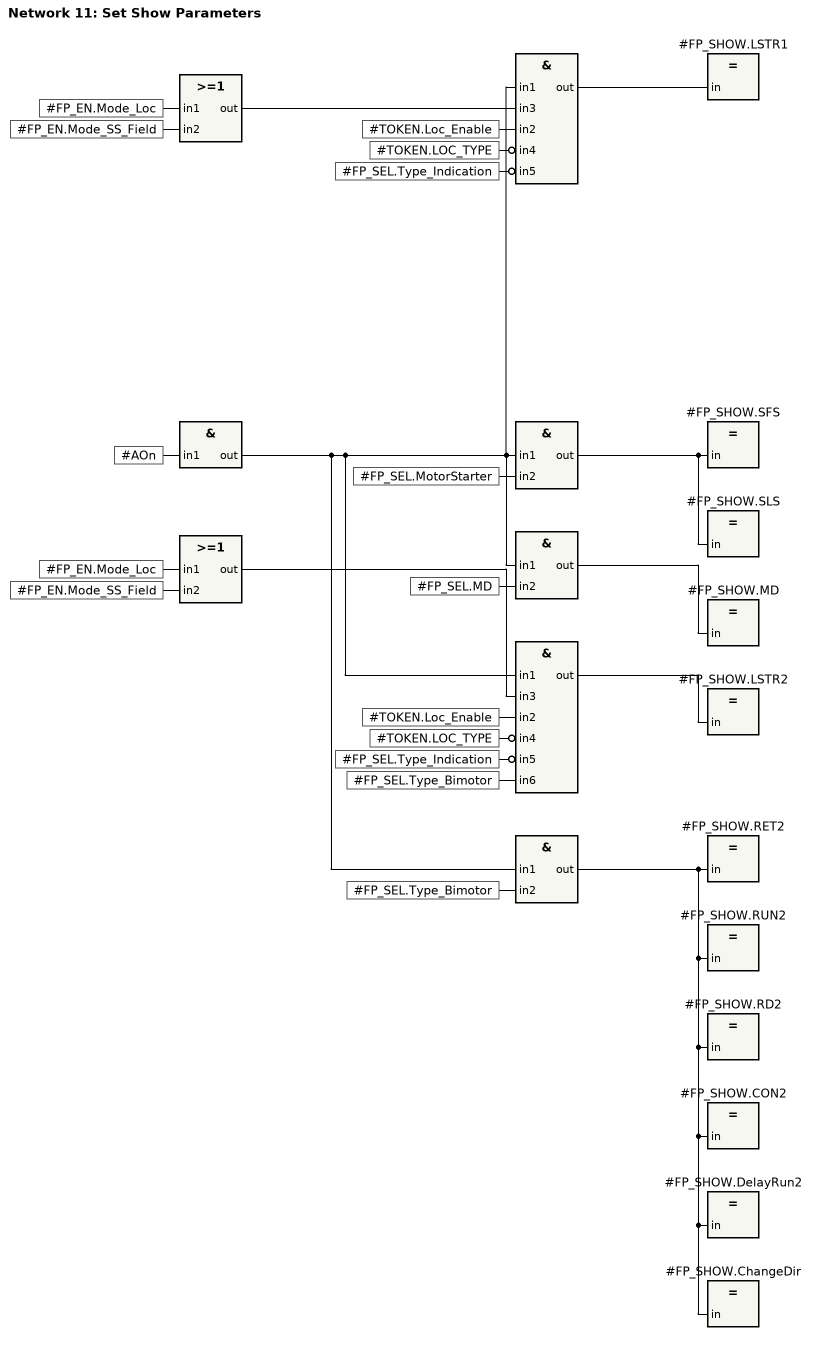
   #FP_SHOW.SFS := #AOn AND #FP_SEL.MotorStarter;
   #FP_SHOW.SLS := #FP_SHOW.SFS;
   #FP_SHOW.MD := #AOn AND #FP_SEL.MD;
   #FP_SHOW.LSTR1 := #AOn AND (#FP_EN.Mode_Loc OR #FP_EN.Mode_SS_Field) AND #TOKEN.Loc_Enable AND NOT #TOKEN.LOC_TYPE AND NOT #FP_SEL.Type_Indication;
   #FP_SHOW.LSTR2 := #AOn AND (#FP_EN.Mode_Loc OR #FP_EN.Mode_SS_Field) AND #TOKEN.Loc_Enable AND NOT #TOKEN.LOC_TYPE AND NOT #FP_SEL.Type_Indication AND #FP_SEL.Type_Bimotor;
   #FP_SHOW.RET2 := #AOn AND #FP_SEL.Type_Bimotor;
   #FP_SHOW.RUN2 := #FP_SHOW.RET2;
   #FP_SHOW.RD2 := #FP_SHOW.RET2;
   #FP_SHOW.CON2 := #FP_SHOW.RET2;
   #FP_SHOW.DelayRun2 := #FP_SHOW.RET2;
   #FP_SHOW.ChangeDir := #FP_SHOW.RET2;
END_REGION

REGION Network 12: SELECT
   // Build 003 - 1.July.2019 (EXTBOB): Added logic to prevent group selection interference when motor is running in "electrical" local mode or mode is controlled from the field.
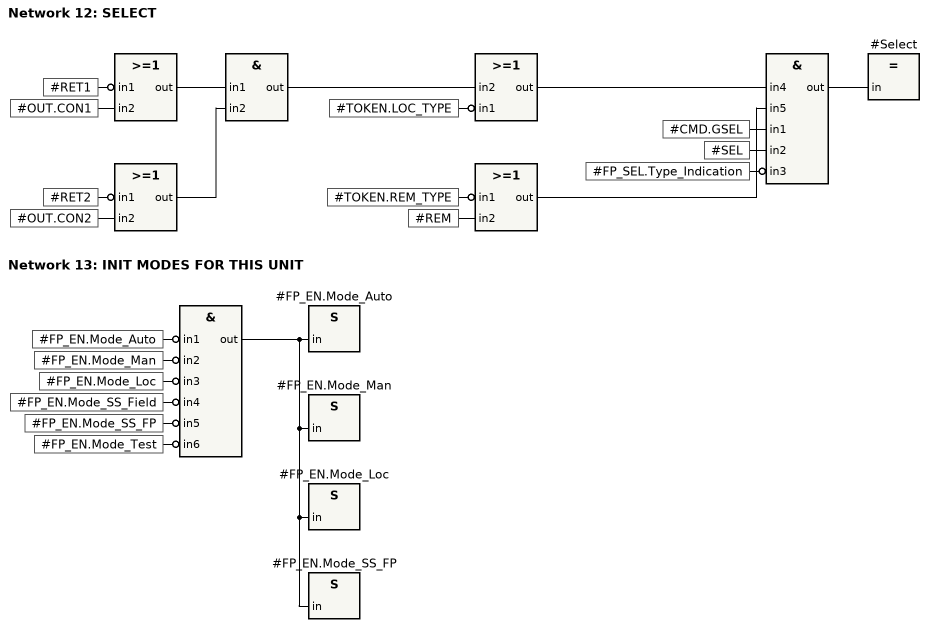
   #Select := (((NOT #RET1 OR #OUT.CON1) AND (NOT #RET2 OR #OUT.CON2)) OR NOT #TOKEN.LOC_TYPE) AND (NOT #TOKEN.REM_TYPE OR #REM) AND #CMD.GSEL AND #SEL AND NOT #FP_SEL.Type_Indication;
END_REGION

REGION Network 13: INIT MODES FOR THIS UNIT
   #_w1 := NOT #FP_EN.Mode_Auto AND NOT #FP_EN.Mode_Man AND NOT #FP_EN.Mode_Loc AND NOT #FP_EN.Mode_SS_Field AND NOT #FP_EN.Mode_SS_FP AND NOT #FP_EN.Mode_Test;
   IF #_w1 THEN
       #FP_EN.Mode_Auto := TRUE;
       #FP_EN.Mode_Man := TRUE;
       #FP_EN.Mode_Loc := TRUE;
       #FP_EN.Mode_SS_FP := TRUE;
   END_IF;
END_REGION

REGION Network 14: SHOW PUSH BUTTONS ON FACEPLATE
   // Build 002 - 25 March 2019 : Loc_type flag removed from Show_Local flag
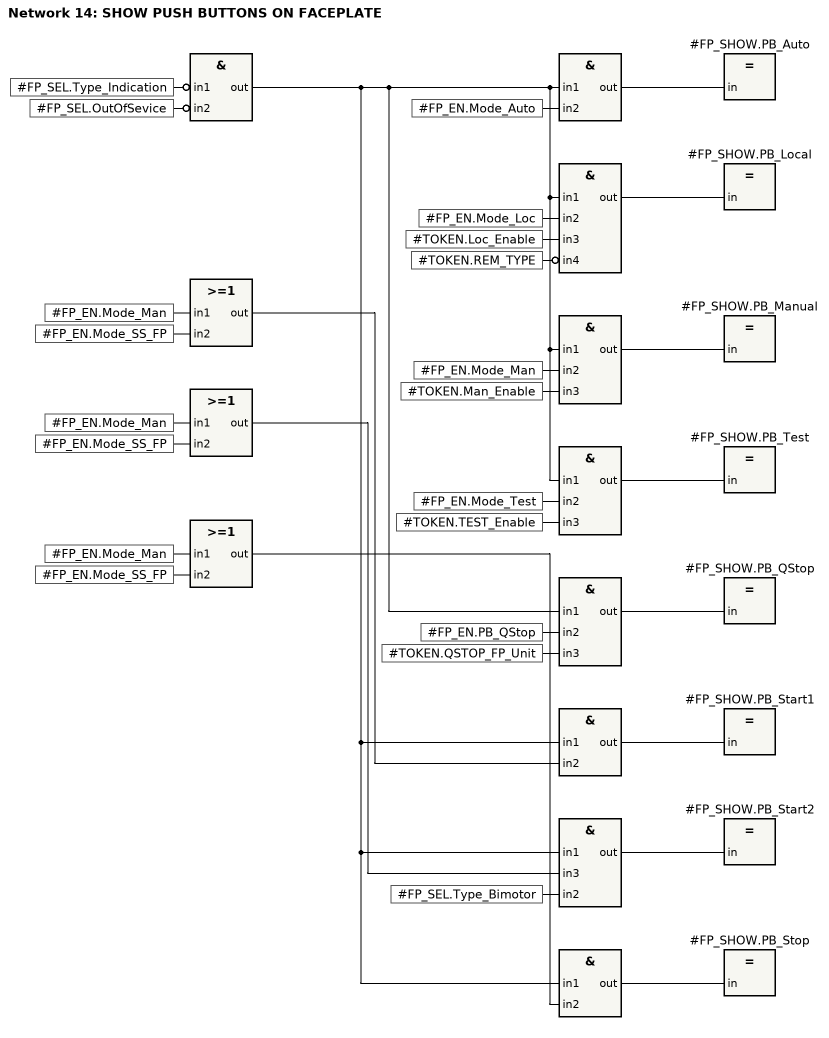
   #_w1 := NOT #FP_SEL.Type_Indication AND NOT #FP_SEL.OutOfSevice;
   #FP_SHOW.PB_Auto := #_w1 AND #FP_EN.Mode_Auto;
   #FP_SHOW.PB_Local := #_w1 AND #FP_EN.Mode_Loc AND #TOKEN.Loc_Enable AND NOT #TOKEN.REM_TYPE;
   #FP_SHOW.PB_Manual := #_w1 AND #FP_EN.Mode_Man AND #TOKEN.Man_Enable;
   #FP_SHOW.PB_Test := #_w1 AND #FP_EN.Mode_Test AND #TOKEN.TEST_Enable;
   #FP_SHOW.PB_QStop := #_w1 AND #FP_EN.PB_QStop AND #TOKEN.QSTOP_FP_Unit;
   #FP_SHOW.PB_Start1 := #_w1 AND (#FP_EN.Mode_Man OR #FP_EN.Mode_SS_FP);
   #FP_SHOW.PB_Start2 := #_w1 AND (#FP_EN.Mode_Man OR #FP_EN.Mode_SS_FP) AND #FP_SEL.Type_Bimotor;
   #FP_SHOW.PB_Stop := #_w1 AND (#FP_EN.Mode_Man OR #FP_EN.Mode_SS_FP);
END_REGION

REGION Network 15: DIMOUT AUTO BUTTON ON FACEPLATE
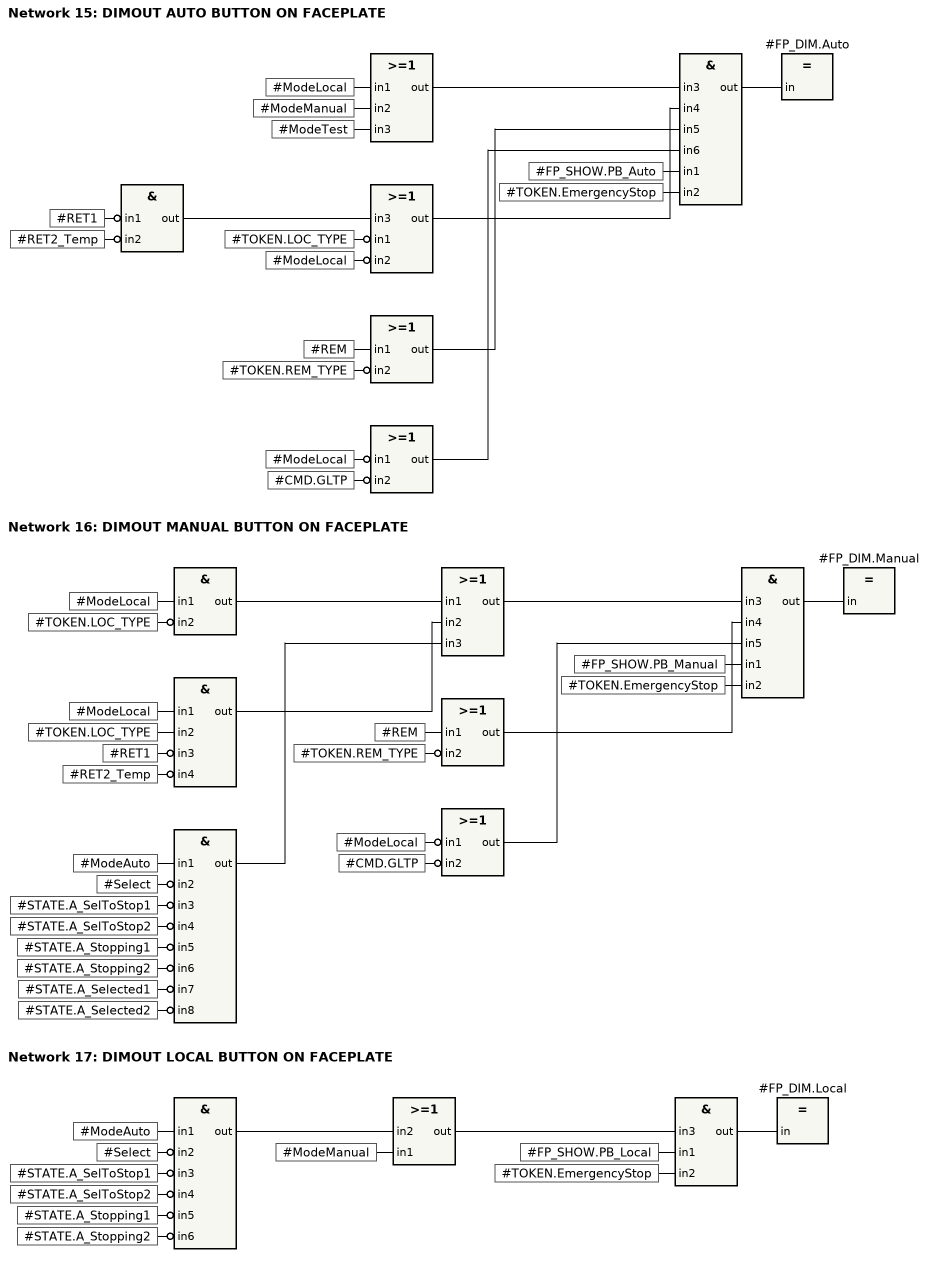
   #FP_DIM.Auto := (#ModeLocal OR #ModeManual OR #ModeTest) AND ((NOT #RET1 AND NOT #RET2_Temp) OR NOT #TOKEN.LOC_TYPE OR NOT #ModeLocal) AND (#REM OR NOT #TOKEN.REM_TYPE) AND (NOT #ModeLocal OR NOT #CMD.GLTP) AND #FP_SHOW.PB_Auto AND #TOKEN.EmergencyStop;
END_REGION

REGION Network 16: DIMOUT MANUAL BUTTON ON FACEPLATE
   #FP_DIM.Manual := ((#ModeLocal AND NOT #TOKEN.LOC_TYPE) OR (#ModeLocal AND #TOKEN.LOC_TYPE AND NOT #RET1 AND NOT #RET2_Temp) OR (#ModeAuto AND NOT #Select AND NOT #STATE.A_SelToStop1 AND NOT #STATE.A_SelToStop2 AND NOT #STATE.A_Stopping1 AND NOT #STATE.A_Stopping2 AND NOT #STATE.A_Selected1 AND NOT #STATE.A_Selected2)) AND (#REM OR NOT #TOKEN.REM_TYPE) AND (NOT #ModeLocal OR NOT #CMD.GLTP) AND #FP_SHOW.PB_Manual AND #TOKEN.EmergencyStop;
END_REGION

REGION Network 17: DIMOUT LOCAL BUTTON ON FACEPLATE
   #FP_DIM.Local := ((#ModeAuto AND NOT #Select AND NOT #STATE.A_SelToStop1 AND NOT #STATE.A_SelToStop2 AND NOT #STATE.A_Stopping1 AND NOT #STATE.A_Stopping2) OR #ModeManual) AND #FP_SHOW.PB_Local AND #TOKEN.EmergencyStop;
END_REGION

REGION Network 18: DIMOUT TEST BUTTON ON FACEPLATE
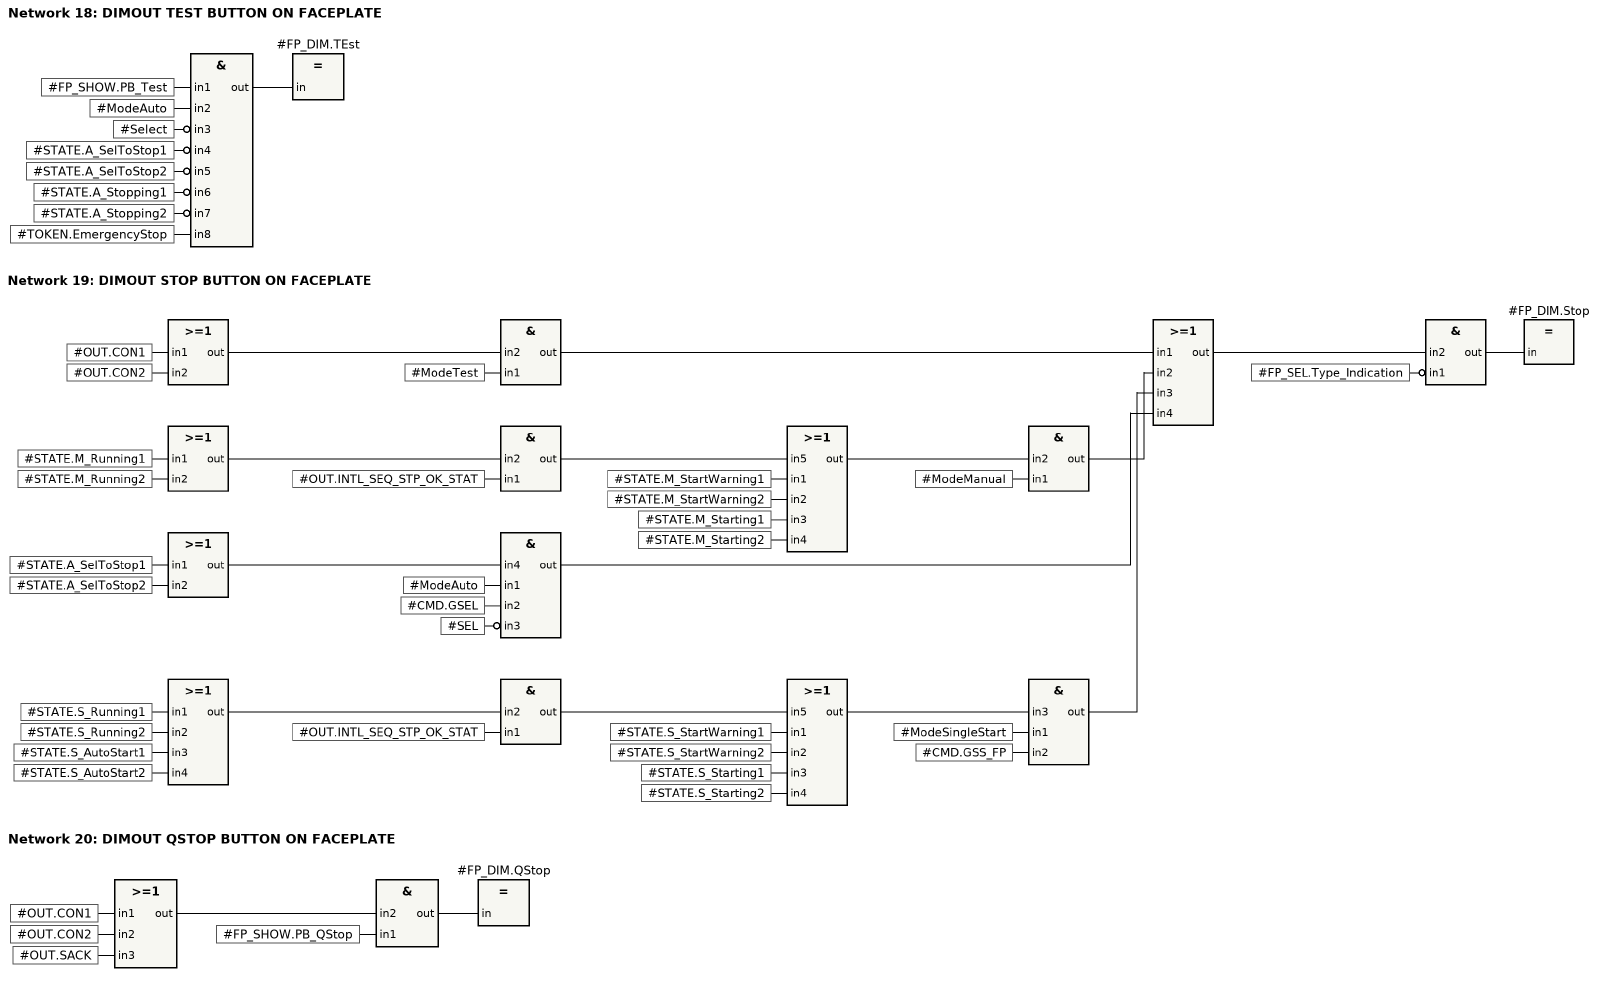
   #FP_DIM.TEst := #FP_SHOW.PB_Test AND #ModeAuto AND NOT #Select AND NOT #STATE.A_SelToStop1 AND NOT #STATE.A_SelToStop2 AND NOT #STATE.A_Stopping1 AND NOT #STATE.A_Stopping2 AND #TOKEN.EmergencyStop;
END_REGION

REGION Network 19: DIMOUT STOP BUTTON ON FACEPLATE
   #FP_DIM.Stop := (((#OUT.CON1 OR #OUT.CON2) AND #ModeTest) OR ((((#STATE.M_Running1 OR #STATE.M_Running2) AND #OUT.INTL_SEQ_STP_OK_STAT) OR #STATE.M_StartWarning1 OR #STATE.M_StartWarning2 OR #STATE.M_Starting1 OR #STATE.M_Starting2) AND #ModeManual) OR ((((#STATE.S_Running1 OR #STATE.S_Running2 OR #STATE.S_AutoStart1 OR #STATE.S_AutoStart2) AND #OUT.INTL_SEQ_STP_OK_STAT) OR #STATE.S_StartWarning1 OR #STATE.S_StartWarning2 OR #STATE.S_Starting1 OR #STATE.S_Starting2) AND #ModeSingleStart AND #CMD.GSS_FP) OR ((#STATE.A_SelToStop1 OR #STATE.A_SelToStop2) AND #ModeAuto AND #CMD.GSEL AND NOT #SEL)) AND NOT #FP_SEL.Type_Indication;
END_REGION

REGION Network 20: DIMOUT QSTOP BUTTON ON FACEPLATE
   #FP_DIM.QStop := (#OUT.CON1 OR #OUT.CON2 OR #OUT.SACK) AND #FP_SHOW.PB_QStop;
END_REGION

REGION Network 21: DIMOUT START1 BUTTON ON FACEPLATE
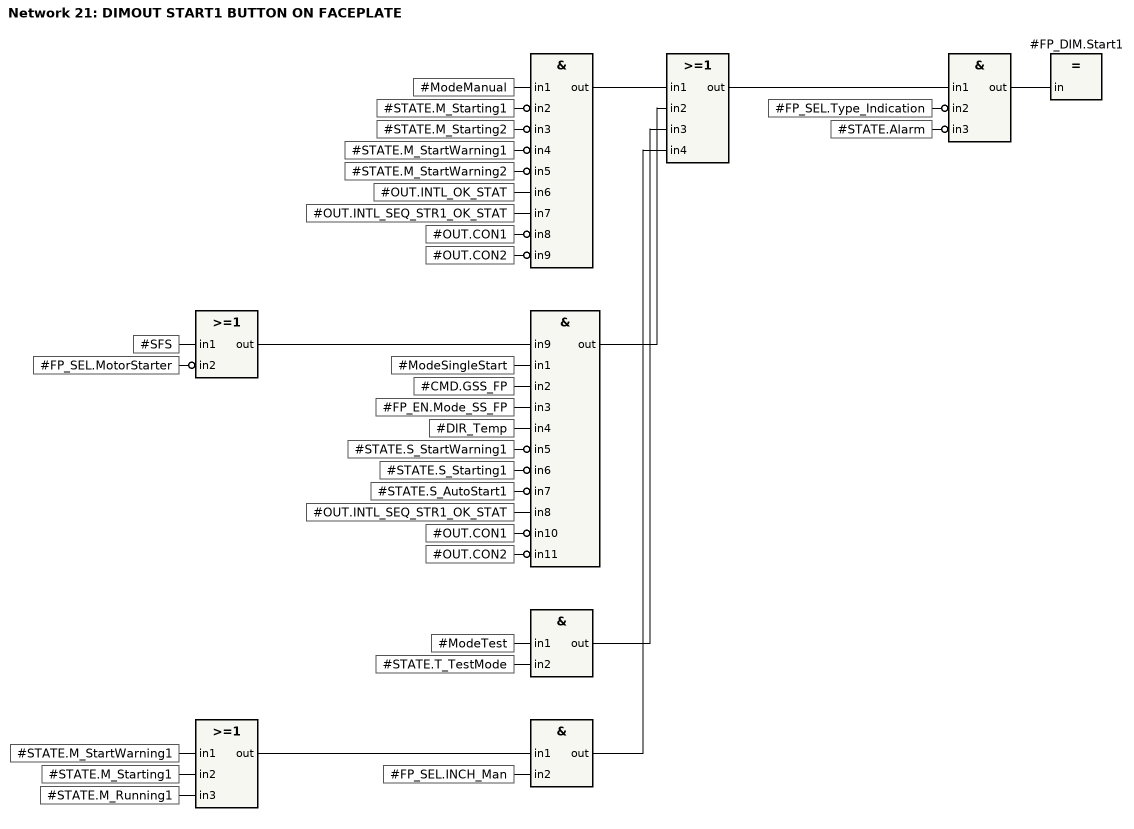
   #FP_DIM.Start1 := ((#ModeManual AND NOT #STATE.M_Starting1 AND NOT #STATE.M_Starting2 AND NOT #STATE.M_StartWarning1 AND NOT #STATE.M_StartWarning2 AND #OUT.INTL_OK_STAT AND #OUT.INTL_SEQ_STR1_OK_STAT AND NOT #OUT.CON1 AND NOT #OUT.CON2) OR ((#SFS OR NOT #FP_SEL.MotorStarter) AND #ModeSingleStart AND #CMD.GSS_FP AND #FP_EN.Mode_SS_FP AND #DIR_Temp AND NOT #STATE.S_StartWarning1 AND NOT #STATE.S_Starting1 AND NOT #STATE.S_AutoStart1 AND #OUT.INTL_SEQ_STR1_OK_STAT AND NOT #OUT.CON1 AND NOT #OUT.CON2) OR (#ModeTest AND #STATE.T_TestMode) OR ((#STATE.M_StartWarning1 OR #STATE.M_Starting1 OR #STATE.M_Running1) AND #FP_SEL.INCH_Man)) AND NOT #FP_SEL.Type_Indication AND NOT #STATE.Alarm;
END_REGION

REGION Network 22: DIMOUT START2 BUTTON ON FACEPLATE
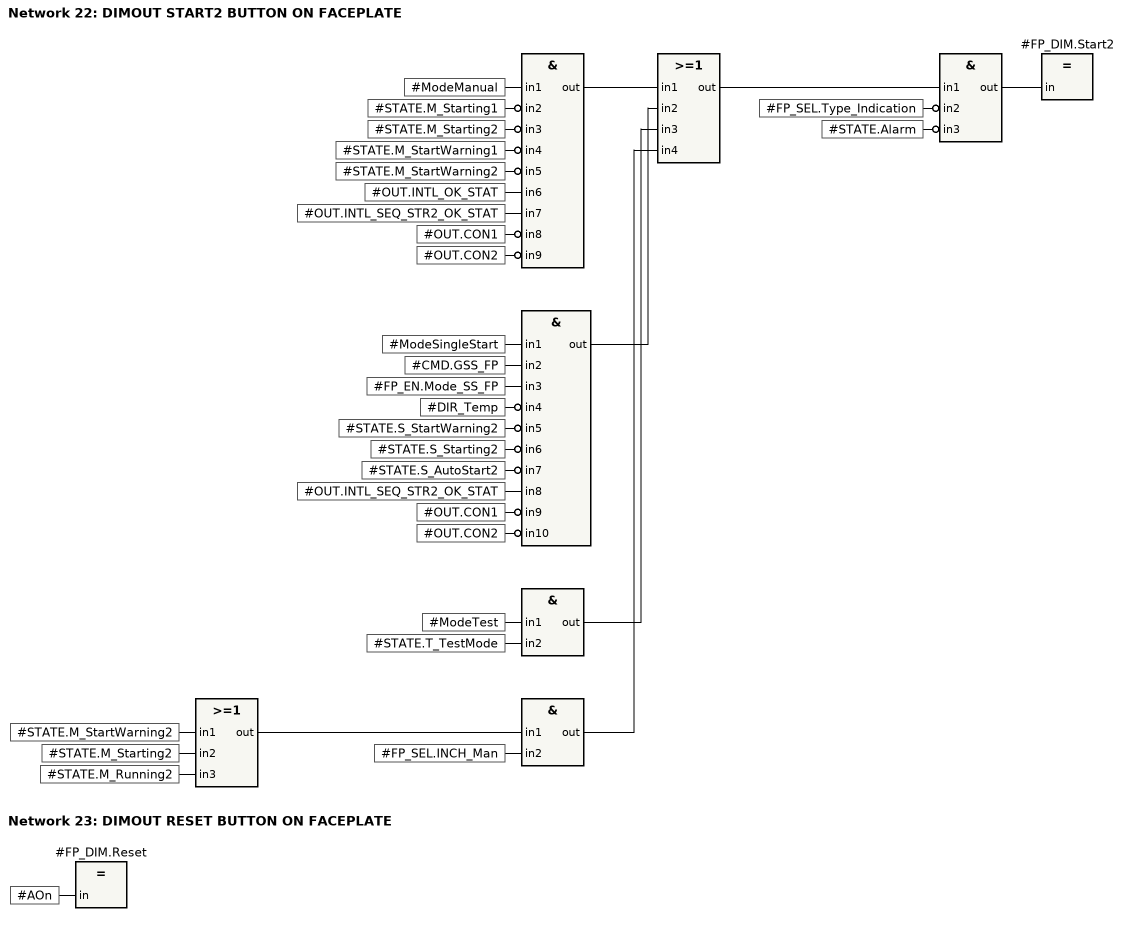
   #FP_DIM.Start2 := ((#ModeManual AND NOT #STATE.M_Starting1 AND NOT #STATE.M_Starting2 AND NOT #STATE.M_StartWarning1 AND NOT #STATE.M_StartWarning2 AND #OUT.INTL_OK_STAT AND #OUT.INTL_SEQ_STR2_OK_STAT AND NOT #OUT.CON1 AND NOT #OUT.CON2) OR (#ModeSingleStart AND #CMD.GSS_FP AND #FP_EN.Mode_SS_FP AND NOT #DIR_Temp AND NOT #STATE.S_StartWarning2 AND NOT #STATE.S_Starting2 AND NOT #STATE.S_AutoStart2 AND #OUT.INTL_SEQ_STR2_OK_STAT AND NOT #OUT.CON1 AND NOT #OUT.CON2) OR (#ModeTest AND #STATE.T_TestMode) OR ((#STATE.M_StartWarning2 OR #STATE.M_Starting2 OR #STATE.M_Running2) AND #FP_SEL.INCH_Man)) AND NOT #FP_SEL.Type_Indication AND NOT #STATE.Alarm;
END_REGION

REGION Network 23: DIMOUT RESET BUTTON ON FACEPLATE
   #FP_DIM.Reset := #AOn;
END_REGION

REGION Network 24: Auto Mode
   // Build 002 - 25 March 2019 : REM flag removed from Modelocal FP_CMD_Auto command
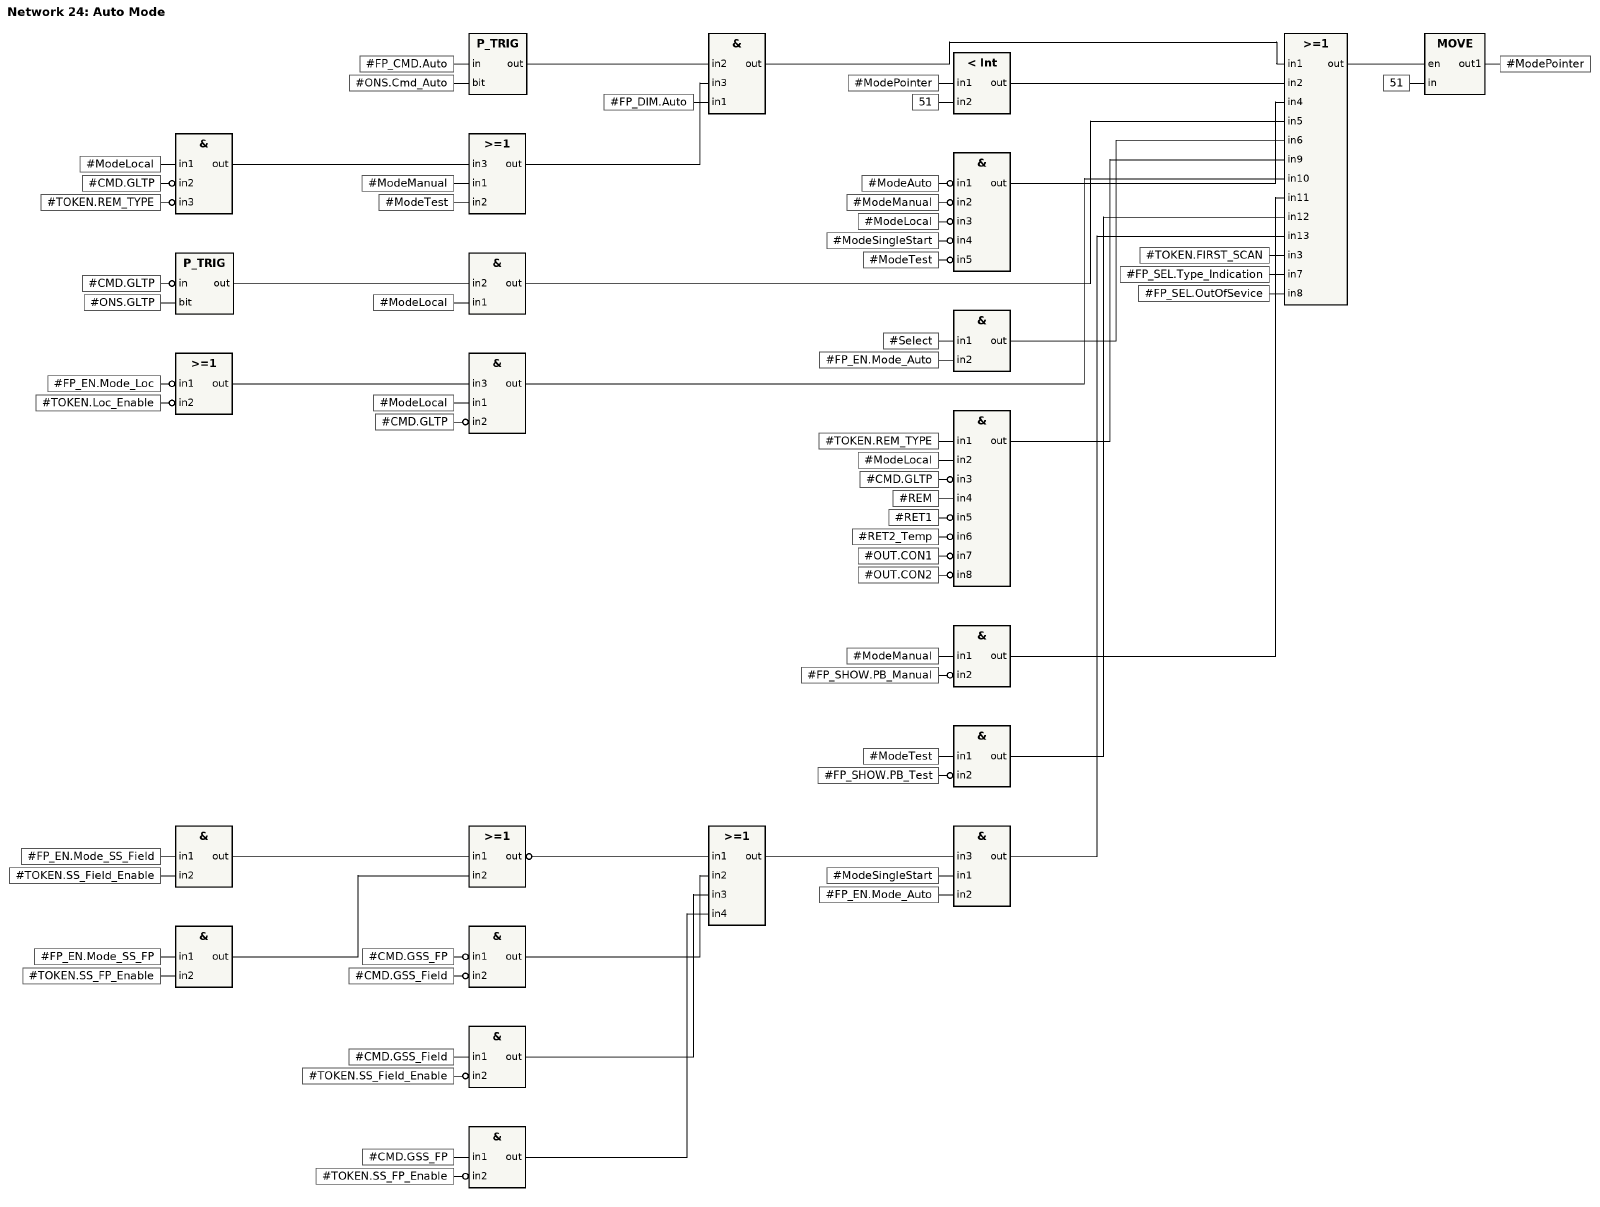
   #_w1 := #FP_CMD.Auto AND NOT #ONS.Cmd_Auto;   // rising edge
   #ONS.Cmd_Auto := #FP_CMD.Auto;
   #_w2 := NOT #CMD.GLTP AND NOT #ONS.GLTP;   // rising edge
   #ONS.GLTP := NOT #CMD.GLTP;
   IF (#_w1 AND ((#ModeLocal AND NOT #CMD.GLTP AND NOT #TOKEN.REM_TYPE) OR #ModeManual OR #ModeTest) AND #FP_DIM.Auto) OR (#ModePointer < 51) OR (NOT #ModeAuto AND NOT #ModeManual AND NOT #ModeLocal AND NOT #ModeSingleStart AND NOT #ModeTest) OR (#_w2 AND #ModeLocal) OR (#Select AND #FP_EN.Mode_Auto) OR (#TOKEN.REM_TYPE AND #ModeLocal AND NOT #CMD.GLTP AND #REM AND NOT #RET1 AND NOT #RET2_Temp AND NOT #OUT.CON1 AND NOT #OUT.CON2) OR ((NOT #FP_EN.Mode_Loc OR NOT #TOKEN.Loc_Enable) AND #ModeLocal AND NOT #CMD.GLTP) OR (#ModeManual AND NOT #FP_SHOW.PB_Manual) OR (#ModeTest AND NOT #FP_SHOW.PB_Test) OR ((NOT ((#FP_EN.Mode_SS_Field AND #TOKEN.SS_Field_Enable) OR (#FP_EN.Mode_SS_FP AND #TOKEN.SS_FP_Enable)) OR (NOT #CMD.GSS_FP AND NOT #CMD.GSS_Field) OR (#CMD.GSS_Field AND NOT #TOKEN.SS_Field_Enable) OR (#CMD.GSS_FP AND NOT #TOKEN.SS_FP_Enable)) AND #ModeSingleStart AND #FP_EN.Mode_Auto) OR #TOKEN.FIRST_SCAN OR #FP_SEL.Type_Indication OR #FP_SEL.OutOfSevice THEN
       #ModePointer := 51;
   END_IF;
END_REGION

REGION Network 25: Mode Manual
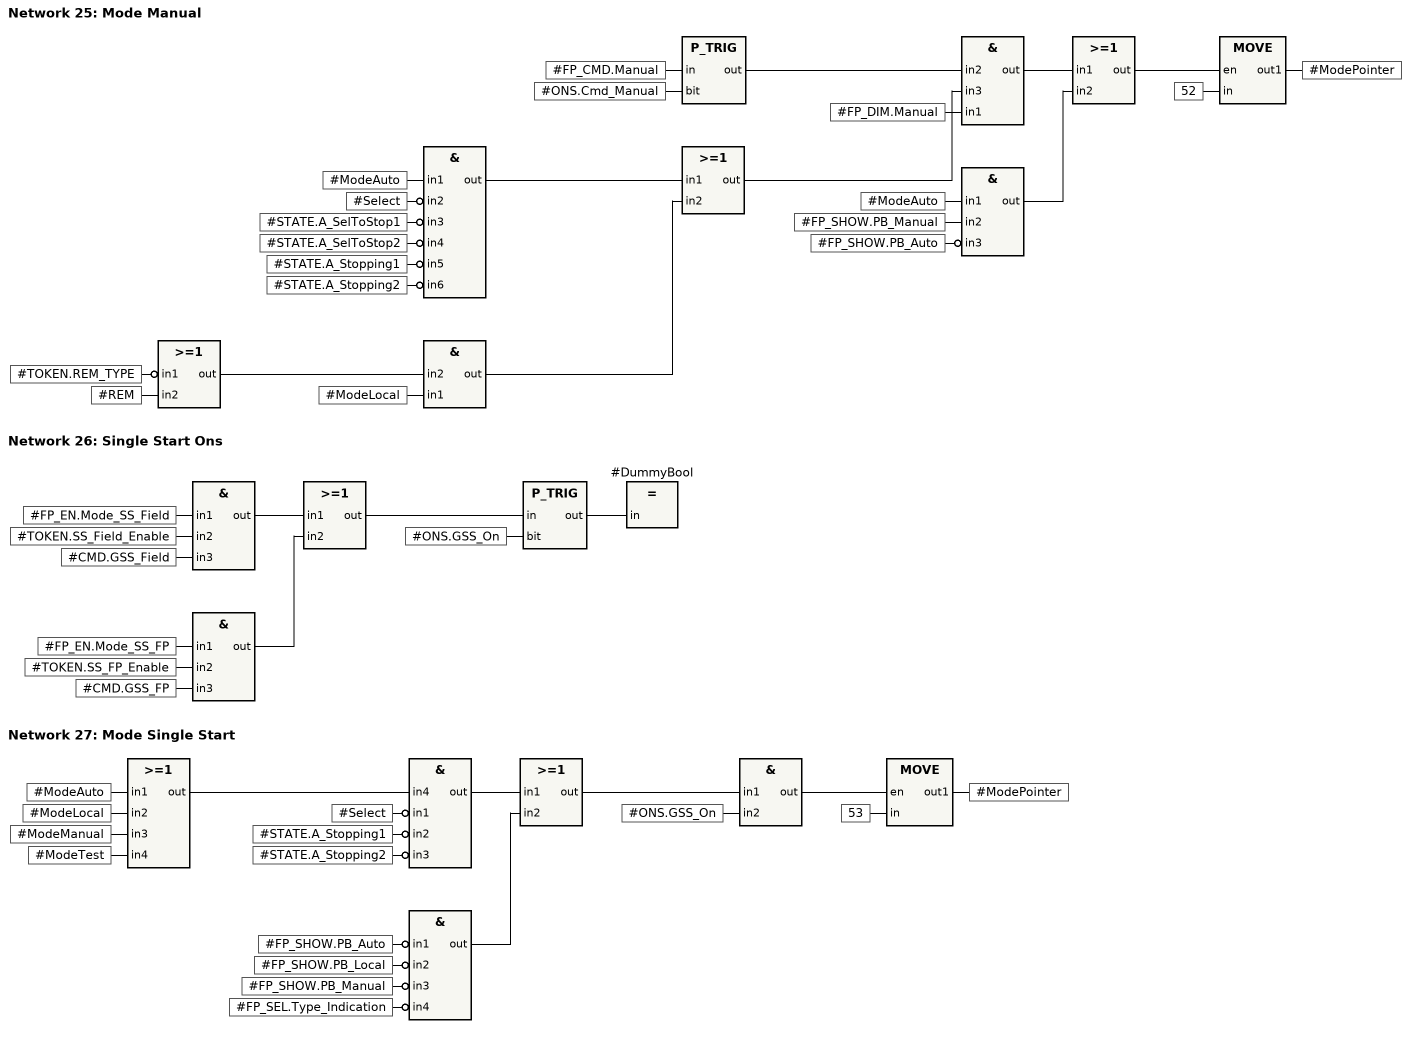
   #_w1 := #FP_CMD.Manual AND NOT #ONS.Cmd_Manual;   // rising edge
   #ONS.Cmd_Manual := #FP_CMD.Manual;
   IF (#_w1 AND ((#ModeAuto AND NOT #Select AND NOT #STATE.A_SelToStop1 AND NOT #STATE.A_SelToStop2 AND NOT #STATE.A_Stopping1 AND NOT #STATE.A_Stopping2) OR ((NOT #TOKEN.REM_TYPE OR #REM) AND #ModeLocal)) AND #FP_DIM.Manual) OR (#ModeAuto AND #FP_SHOW.PB_Manual AND NOT #FP_SHOW.PB_Auto) THEN
       #ModePointer := 52;
   END_IF;
END_REGION

REGION Network 26: Single Start Ons
   // Build 003 - 1.July.2019 (EXTBOB): Added ONS and Created New Network to separate trigger from pre-conditions
   #_w1 := (#FP_EN.Mode_SS_Field AND #TOKEN.SS_Field_Enable AND #CMD.GSS_Field) OR (#FP_EN.Mode_SS_FP AND #TOKEN.SS_FP_Enable AND #CMD.GSS_FP);
   #_w2 := #_w1 AND NOT #ONS.GSS_On;   // rising edge
   #ONS.GSS_On := #_w1;
   #DummyBool := #_w2;
END_REGION

REGION Network 27: Mode Single Start
   // Build 003 - 1.July.2019 (EXTBOB): Added Single Start ONS and Removed the Single start trigger condition & made as seperate Network above
   IF (((#ModeAuto OR #ModeLocal OR #ModeManual OR #ModeTest) AND NOT #Select AND NOT #STATE.A_Stopping1 AND NOT #STATE.A_Stopping2) OR (NOT #FP_SHOW.PB_Auto AND NOT #FP_SHOW.PB_Local AND NOT #FP_SHOW.PB_Manual AND NOT #FP_SEL.Type_Indication)) AND #ONS.GSS_On THEN
       #ModePointer := 53;
   END_IF;
END_REGION

REGION Network 28: Mode Local
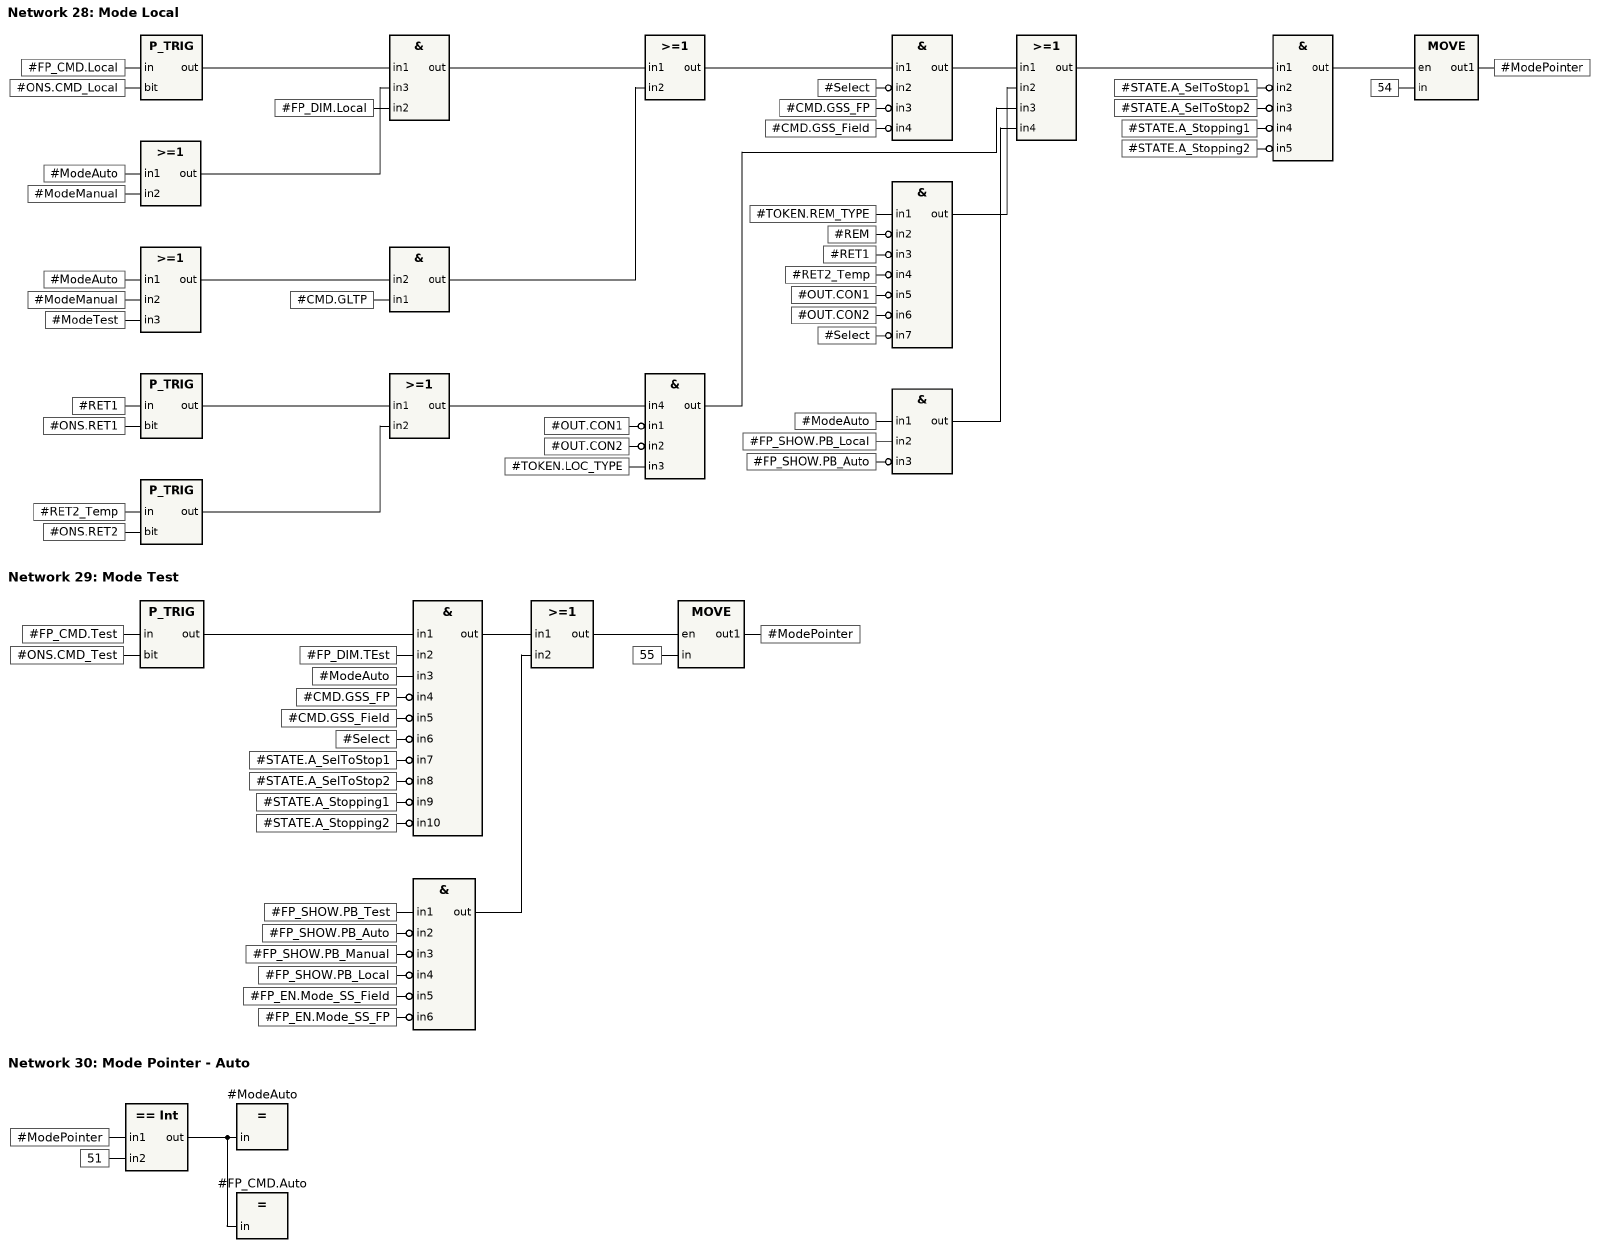
   #_w1 := #FP_CMD.Local AND NOT #ONS.CMD_Local;   // rising edge
   #ONS.CMD_Local := #FP_CMD.Local;
   #_w2 := #RET1 AND NOT #ONS.RET1;   // rising edge
   #ONS.RET1 := #RET1;
   #_w3 := #RET2_Temp AND NOT #ONS.RET2;   // rising edge
   #ONS.RET2 := #RET2_Temp;
   IF ((((#_w1 AND (#ModeAuto OR #ModeManual) AND #FP_DIM.Local) OR ((#ModeAuto OR #ModeManual OR #ModeTest) AND #CMD.GLTP)) AND NOT #Select AND NOT #CMD.GSS_FP AND NOT #CMD.GSS_Field) OR (#TOKEN.REM_TYPE AND NOT #REM AND NOT #RET1 AND NOT #RET2_Temp AND NOT #OUT.CON1 AND NOT #OUT.CON2 AND NOT #Select) OR ((#_w2 OR #_w3) AND NOT #OUT.CON1 AND NOT #OUT.CON2 AND #TOKEN.LOC_TYPE) OR (#ModeAuto AND #FP_SHOW.PB_Local AND NOT #FP_SHOW.PB_Auto)) AND NOT #STATE.A_SelToStop1 AND NOT #STATE.A_SelToStop2 AND NOT #STATE.A_Stopping1 AND NOT #STATE.A_Stopping2 THEN
       #ModePointer := 54;
   END_IF;
END_REGION

REGION Network 29: Mode Test
   #_w1 := #FP_CMD.Test AND NOT #ONS.CMD_Test;   // rising edge
   #ONS.CMD_Test := #FP_CMD.Test;
   IF (#_w1 AND #FP_DIM.TEst AND #ModeAuto AND NOT #CMD.GSS_FP AND NOT #CMD.GSS_Field AND NOT #Select AND NOT #STATE.A_SelToStop1 AND NOT #STATE.A_SelToStop2 AND NOT #STATE.A_Stopping1 AND NOT #STATE.A_Stopping2) OR (#FP_SHOW.PB_Test AND NOT #FP_SHOW.PB_Auto AND NOT #FP_SHOW.PB_Manual AND NOT #FP_SHOW.PB_Local AND NOT #FP_EN.Mode_SS_Field AND NOT #FP_EN.Mode_SS_FP) THEN
       #ModePointer := 55;
   END_IF;
END_REGION

REGION Network 30: Mode Pointer - Auto
   #ModeAuto := #ModePointer = 51;
   #FP_CMD.Auto := #ModeAuto;
END_REGION

REGION Network 31: Mode Pointer - Manual
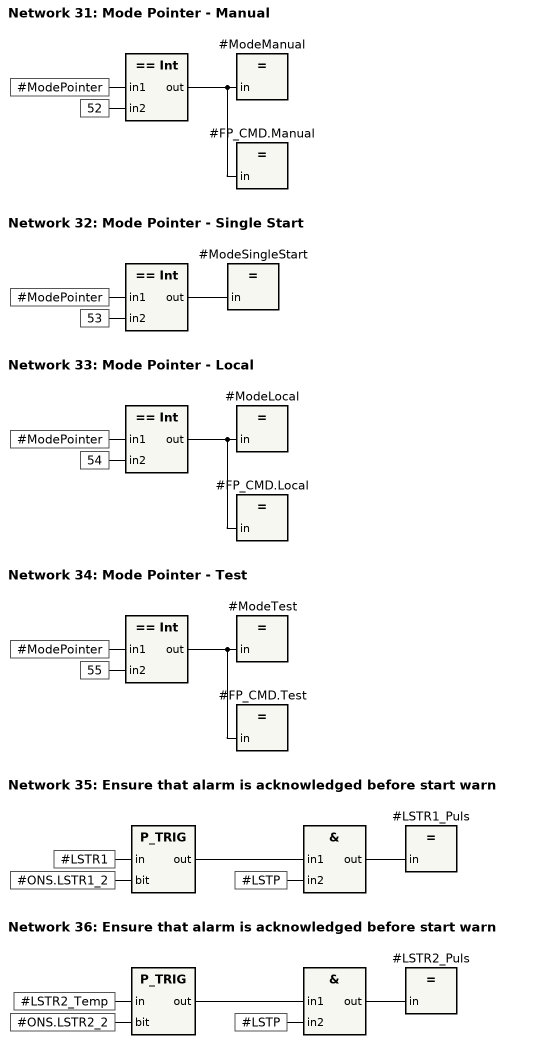
   #ModeManual := #ModePointer = 52;
   #FP_CMD.Manual := #ModeManual;
END_REGION

REGION Network 32: Mode Pointer - Single Start
   #ModeSingleStart := #ModePointer = 53;
END_REGION

REGION Network 33: Mode Pointer - Local
   #ModeLocal := #ModePointer = 54;
   #FP_CMD.Local := #ModeLocal;
END_REGION

REGION Network 34: Mode Pointer - Test
   #ModeTest := #ModePointer = 55;
   #FP_CMD.Test := #ModeTest;
END_REGION

REGION Network 35: Ensure that alarm is acknowledged before start warn
   // Build 003 - 30 Jun 2019 (EXTBOB): Added LSTP to prevent pulse output
   #_w1 := #LSTR1 AND NOT #ONS.LSTR1_2;   // rising edge
   #ONS.LSTR1_2 := #LSTR1;
   #LSTR1_Puls := #_w1 AND #LSTP;
END_REGION

REGION Network 36: Ensure that alarm is acknowledged before start warn
   // Build 003 - 30 Jun 2019 (EXTBOB): Added LSTP to prevent pulse output
   #_w1 := #LSTR2_Temp AND NOT #ONS.LSTR2_2;   // rising edge
   #ONS.LSTR2_2 := #LSTR2_Temp;
   #LSTR2_Puls := #_w1 AND #LSTP;
END_REGION

REGION Network 37: FACEPLATE COMMANDS (Pulse Type)
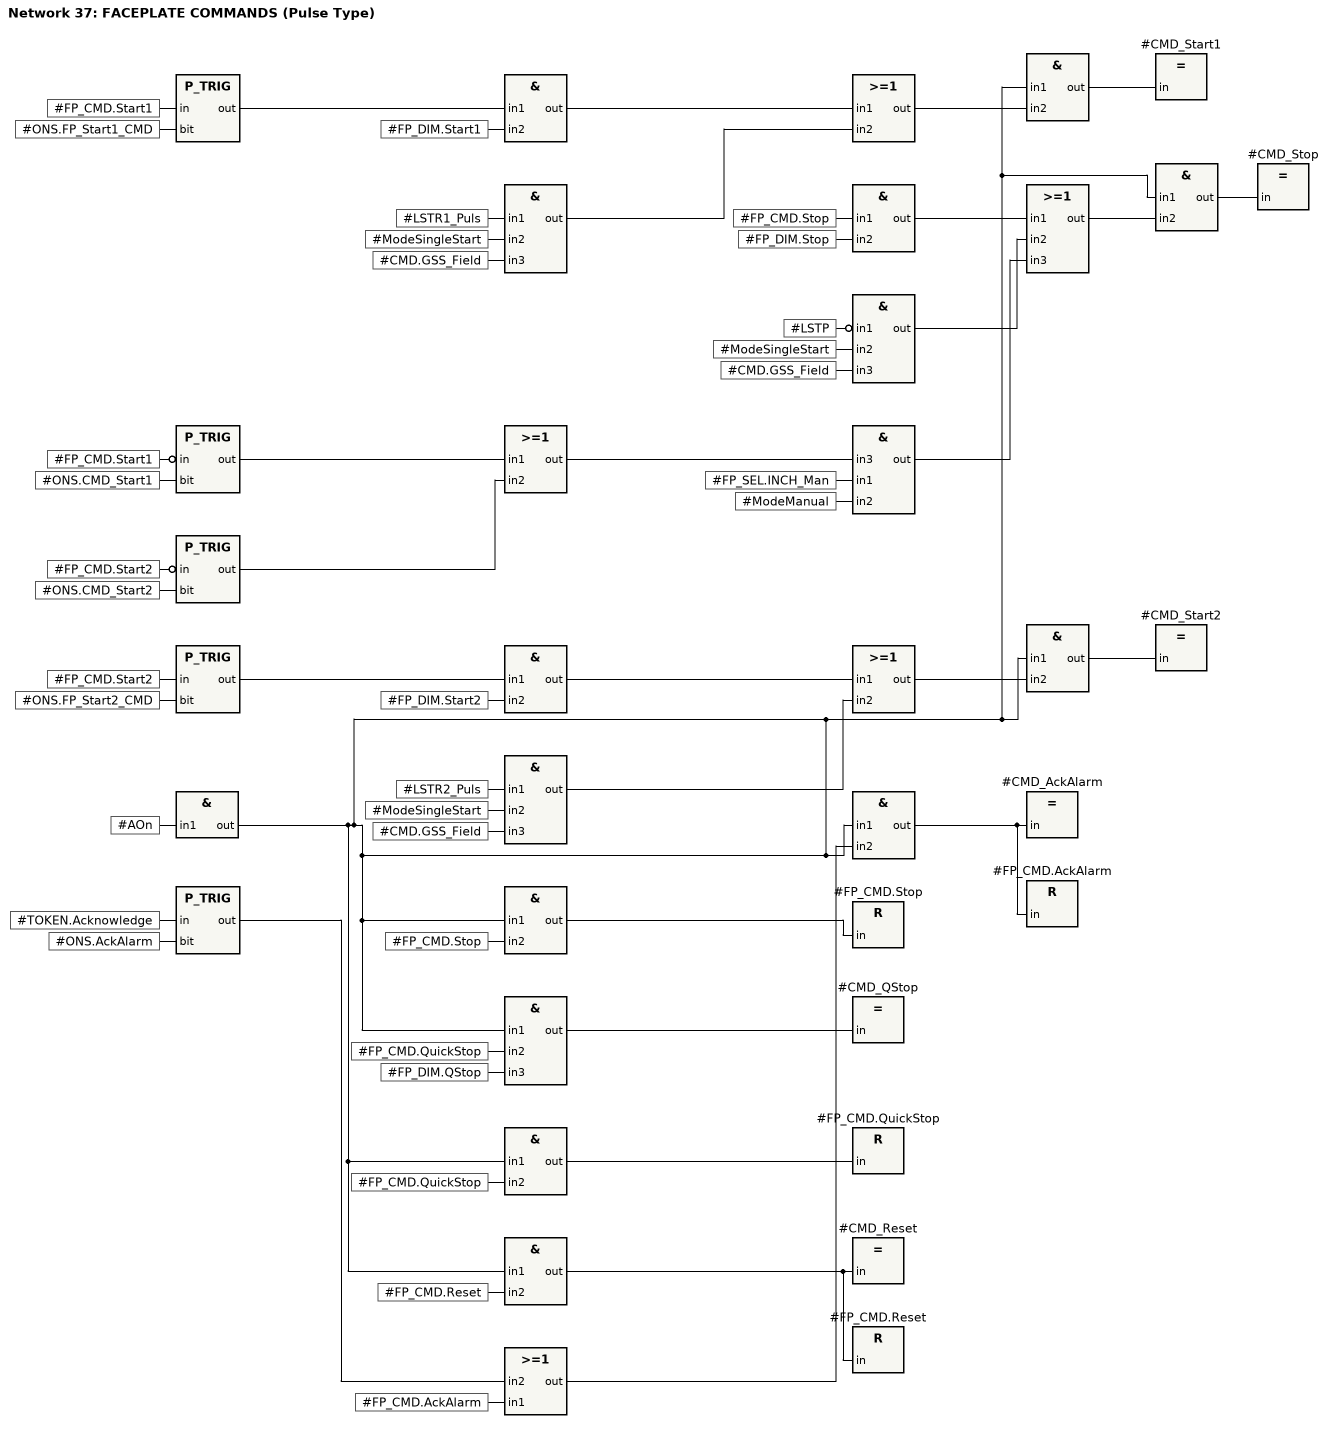
   #_w1 := #FP_CMD.Start1 AND NOT #ONS.FP_Start1_CMD;   // rising edge
   #ONS.FP_Start1_CMD := #FP_CMD.Start1;
   #CMD_Start1 := #AOn AND ((#_w1 AND #FP_DIM.Start1) OR (#LSTR1_Puls AND #ModeSingleStart AND #CMD.GSS_Field));
   #_w2 := #FP_CMD.Start2 AND NOT #ONS.FP_Start2_CMD;   // rising edge
   #ONS.FP_Start2_CMD := #FP_CMD.Start2;
   #CMD_Start2 := #AOn AND ((#_w2 AND #FP_DIM.Start2) OR (#LSTR2_Puls AND #ModeSingleStart AND #CMD.GSS_Field));
   #_w3 := NOT #FP_CMD.Start1 AND NOT #ONS.CMD_Start1;   // rising edge
   #ONS.CMD_Start1 := NOT #FP_CMD.Start1;
   #_w4 := NOT #FP_CMD.Start2 AND NOT #ONS.CMD_Start2;   // rising edge
   #ONS.CMD_Start2 := NOT #FP_CMD.Start2;
   #CMD_Stop := #AOn AND ((#FP_CMD.Stop AND #FP_DIM.Stop) OR (NOT #LSTP AND #ModeSingleStart AND #CMD.GSS_Field) OR ((#_w3 OR #_w4) AND #FP_SEL.INCH_Man AND #ModeManual));
   IF #AOn AND #FP_CMD.Stop THEN #FP_CMD.Stop := FALSE; END_IF;
   #CMD_QStop := #AOn AND #FP_CMD.QuickStop AND #FP_DIM.QStop;
   IF #AOn AND #FP_CMD.QuickStop THEN #FP_CMD.QuickStop := FALSE; END_IF;
   #CMD_Reset := #AOn AND #FP_CMD.Reset;
   IF #CMD_Reset THEN #FP_CMD.Reset := FALSE; END_IF;
   #_w5 := #TOKEN.Acknowledge AND NOT #ONS.AckAlarm;   // rising edge
   #ONS.AckAlarm := #TOKEN.Acknowledge;
   #CMD_AckAlarm := #AOn AND (#_w5 OR #FP_CMD.AckAlarm);
   IF #CMD_AckAlarm THEN #FP_CMD.AckAlarm := FALSE; END_IF;
END_REGION

REGION Network 38: Command Reset
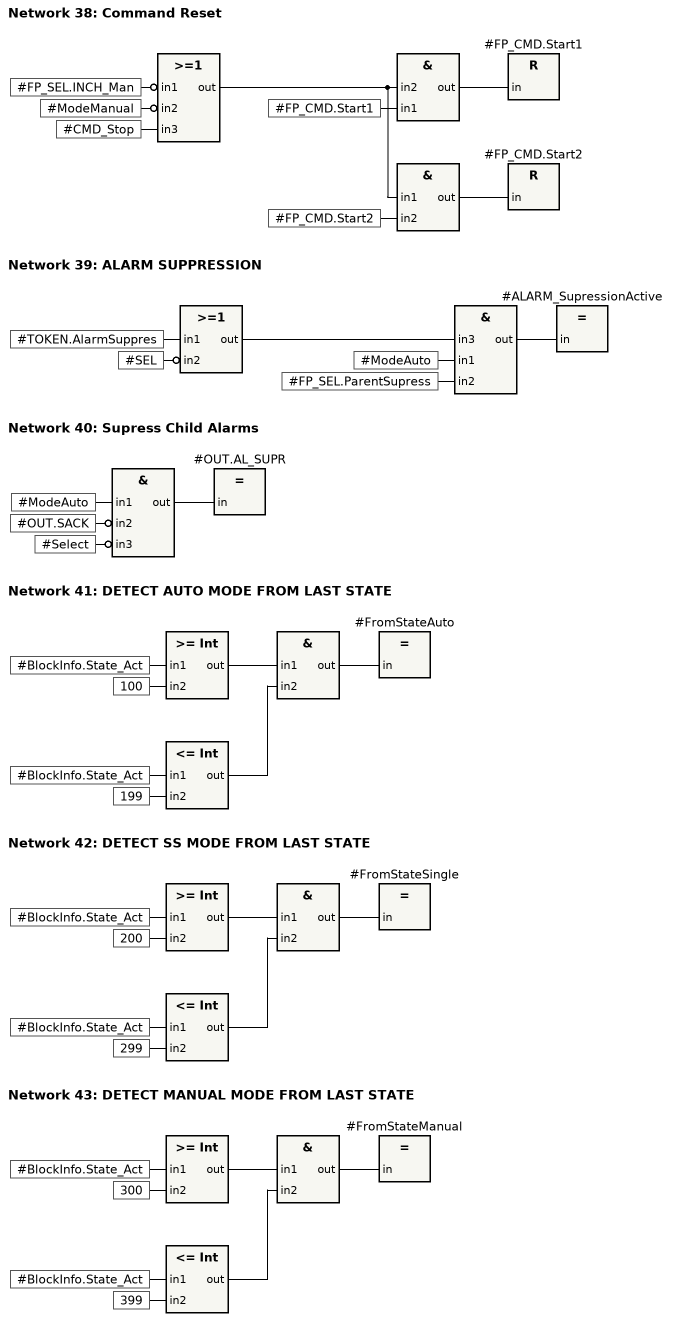
   #_w1 := NOT #FP_SEL.INCH_Man OR NOT #ModeManual OR #CMD_Stop;
   IF #_w1 AND #FP_CMD.Start1 THEN #FP_CMD.Start1 := FALSE; END_IF;
   IF #_w1 AND #FP_CMD.Start2 THEN #FP_CMD.Start2 := FALSE; END_IF;
END_REGION

REGION Network 39: ALARM SUPPRESSION
   #ALARM_SupressionActive := (#TOKEN.AlarmSuppres OR NOT #SEL) AND #ModeAuto AND #FP_SEL.ParentSupress;
END_REGION

REGION Network 40: Supress Child Alarms
   #OUT.AL_SUPR := #ModeAuto AND NOT #OUT.SACK AND NOT #Select;
END_REGION

REGION Network 41: DETECT AUTO MODE FROM LAST STATE
   #FromStateAuto := (#BlockInfo.State_Act >= 100) AND (#BlockInfo.State_Act <= 199);
END_REGION

REGION Network 42: DETECT SS MODE FROM LAST STATE
   #FromStateSingle := (#BlockInfo.State_Act >= 200) AND (#BlockInfo.State_Act <= 299);
END_REGION

REGION Network 43: DETECT MANUAL MODE FROM LAST STATE
   #FromStateManual := (#BlockInfo.State_Act >= 300) AND (#BlockInfo.State_Act <= 399);
END_REGION

REGION Network 44: DETECT LOCAL MODE FROM LAST STATE
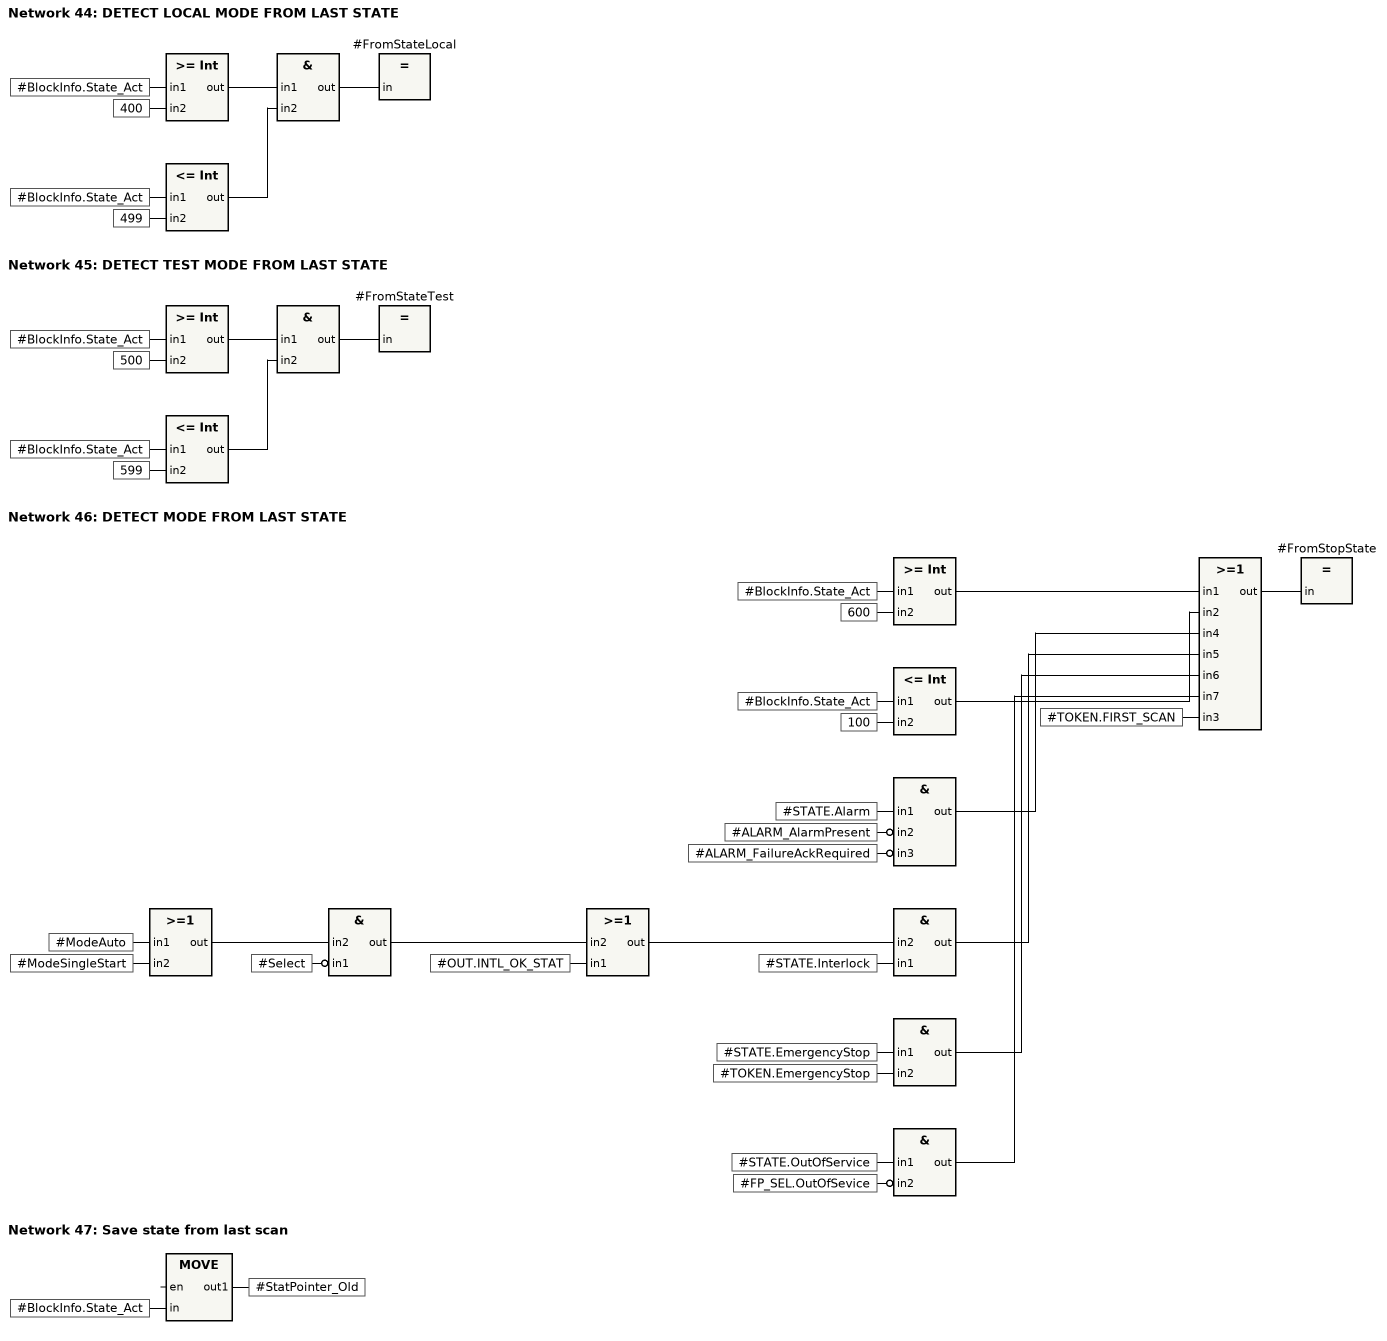
   #FromStateLocal := (#BlockInfo.State_Act >= 400) AND (#BlockInfo.State_Act <= 499);
END_REGION

REGION Network 45: DETECT TEST MODE FROM LAST STATE
   #FromStateTest := (#BlockInfo.State_Act >= 500) AND (#BlockInfo.State_Act <= 599);
END_REGION

REGION Network 46: DETECT MODE FROM LAST STATE
   #FromStopState := (#BlockInfo.State_Act >= 600) OR (#BlockInfo.State_Act <= 100) OR (#STATE.Alarm AND NOT #ALARM_AlarmPresent AND NOT #ALARM_FailureAckRequired) OR ((((#ModeAuto OR #ModeSingleStart) AND NOT #Select) OR #OUT.INTL_OK_STAT) AND #STATE.Interlock) OR (#STATE.EmergencyStop AND #TOKEN.EmergencyStop) OR (#STATE.OutOfService AND NOT #FP_SEL.OutOfSevice) OR #TOKEN.FIRST_SCAN;
END_REGION

REGION Network 47: Save state from last scan
   #StatPointer_Old := #BlockInfo.State_Act;
END_REGION

REGION Network 48
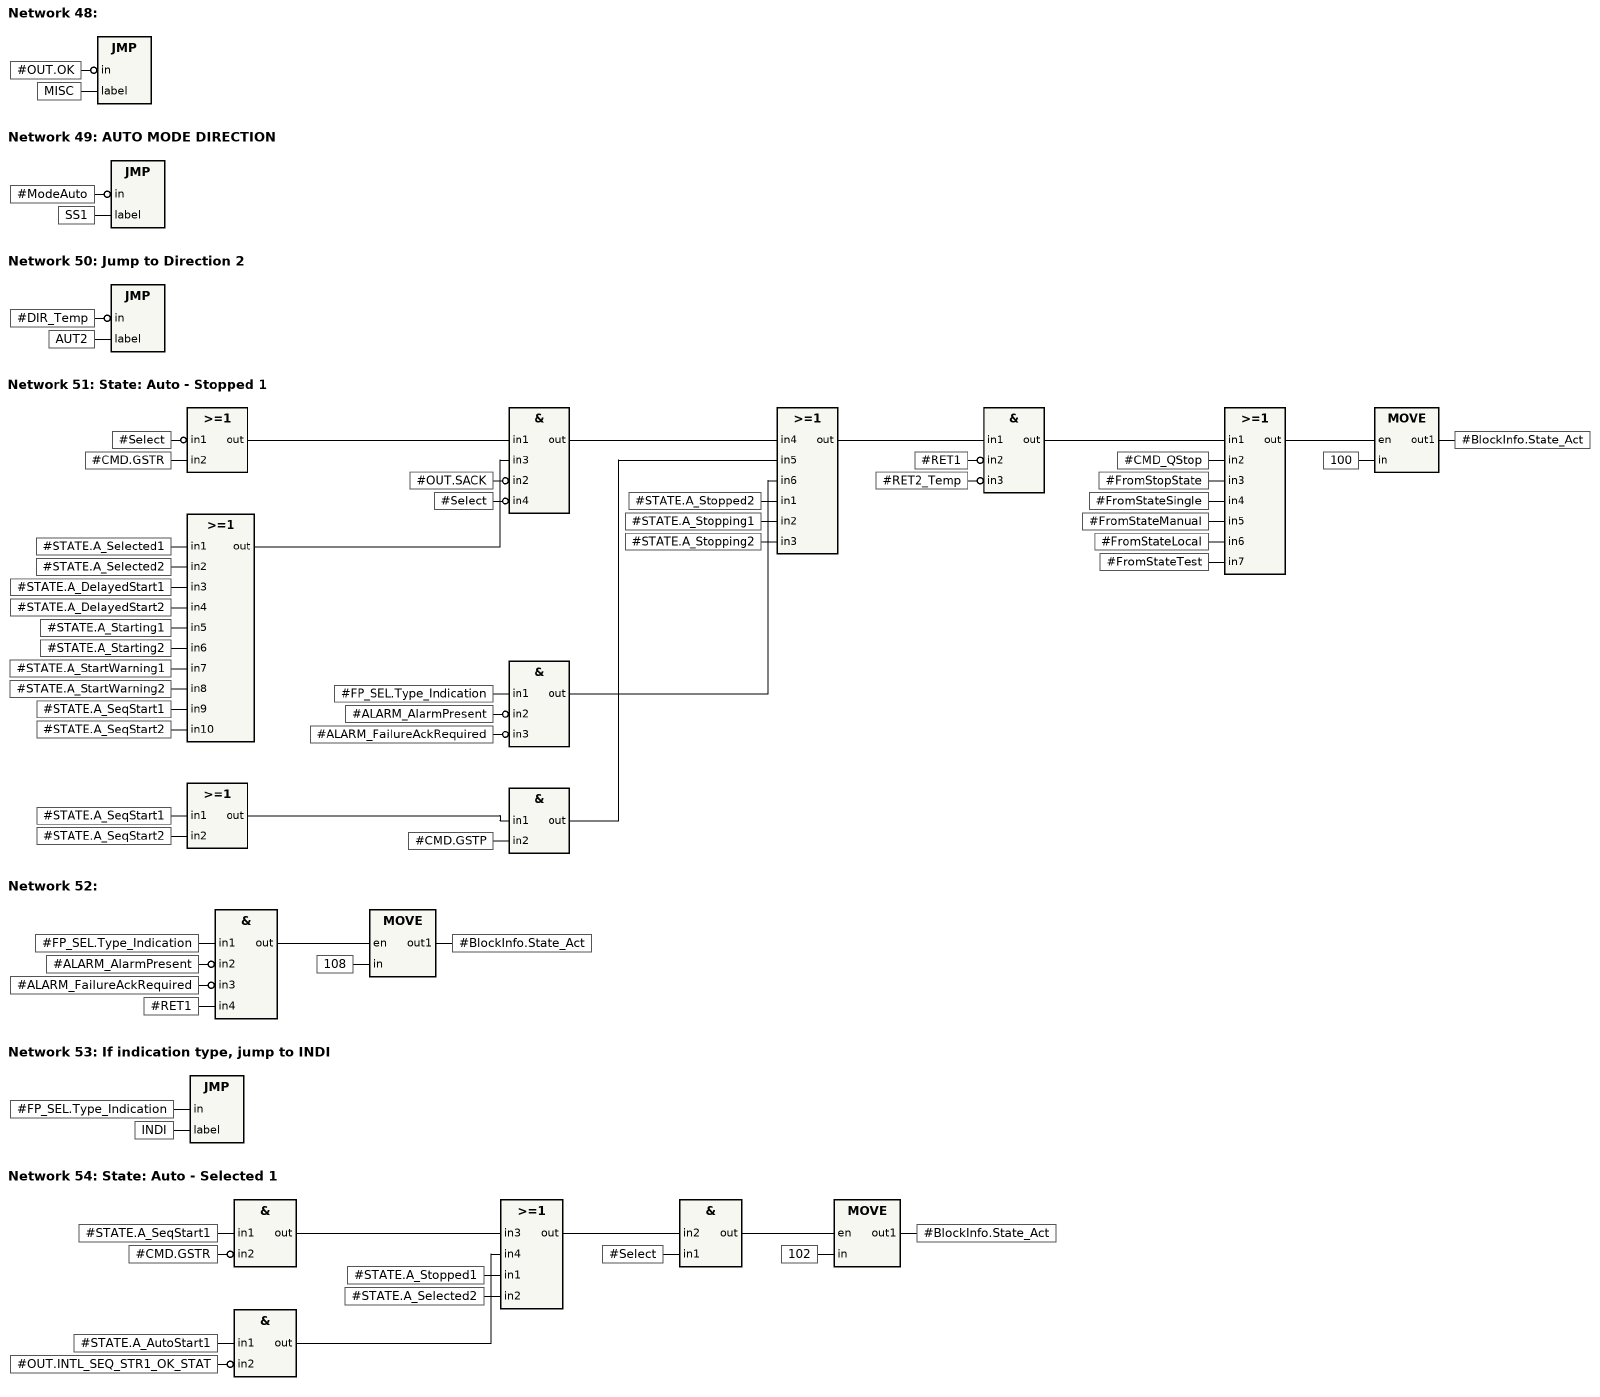
   IF NOT #OUT.OK THEN GOTO MISC; END_IF;
END_REGION

REGION Network 49: AUTO MODE DIRECTION
   IF NOT #ModeAuto THEN GOTO SS1; END_IF;
END_REGION

REGION Network 50: Jump to Direction 2
   IF NOT #DIR_Temp THEN GOTO AUT2; END_IF;
END_REGION

REGION Network 51: State: Auto - Stopped 1
   IF ((((NOT #Select OR #CMD.GSTR) AND (#STATE.A_Selected1 OR #STATE.A_Selected2 OR #STATE.A_DelayedStart1 OR #STATE.A_DelayedStart2 OR #STATE.A_Starting1 OR #STATE.A_Starting2 OR #STATE.A_StartWarning1 OR #STATE.A_StartWarning2 OR #STATE.A_SeqStart1 OR #STATE.A_SeqStart2) AND NOT #OUT.SACK AND NOT #Select) OR ((#STATE.A_SeqStart1 OR #STATE.A_SeqStart2) AND #CMD.GSTP) OR (#FP_SEL.Type_Indication AND NOT #ALARM_AlarmPresent AND NOT #ALARM_FailureAckRequired) OR #STATE.A_Stopped2 OR #STATE.A_Stopping1 OR #STATE.A_Stopping2) AND NOT #RET1 AND NOT #RET2_Temp) OR #CMD_QStop OR #FromStopState OR #FromStateSingle OR #FromStateManual OR #FromStateLocal OR #FromStateTest THEN
       #BlockInfo.State_Act := 100;
   END_IF;
END_REGION

REGION Network 52
   IF #FP_SEL.Type_Indication AND NOT #ALARM_AlarmPresent AND NOT #ALARM_FailureAckRequired AND #RET1 THEN
       #BlockInfo.State_Act := 108;
   END_IF;
END_REGION

REGION Network 53: If indication type, jump to INDI
   IF #FP_SEL.Type_Indication THEN GOTO INDI; END_IF;
END_REGION

REGION Network 54: State: Auto - Selected 1
   // Build 002 - 25 March 2019 : AutoStart1 with SeqStart Interlock condition added
   IF ((#STATE.A_SeqStart1 AND NOT #CMD.GSTR) OR (#STATE.A_AutoStart1 AND NOT #OUT.INTL_SEQ_STR1_OK_STAT) OR #STATE.A_Stopped1 OR #STATE.A_Selected2) AND #Select THEN
       #BlockInfo.State_Act := 102;
   END_IF;
END_REGION

REGION Network 55: State: Auto - Sequence Start 1
   // Build 006 - 29 Aug 2019 (EXTBOB) : AutoStart flag removed to have wait start state when astr = 0 during group start contion
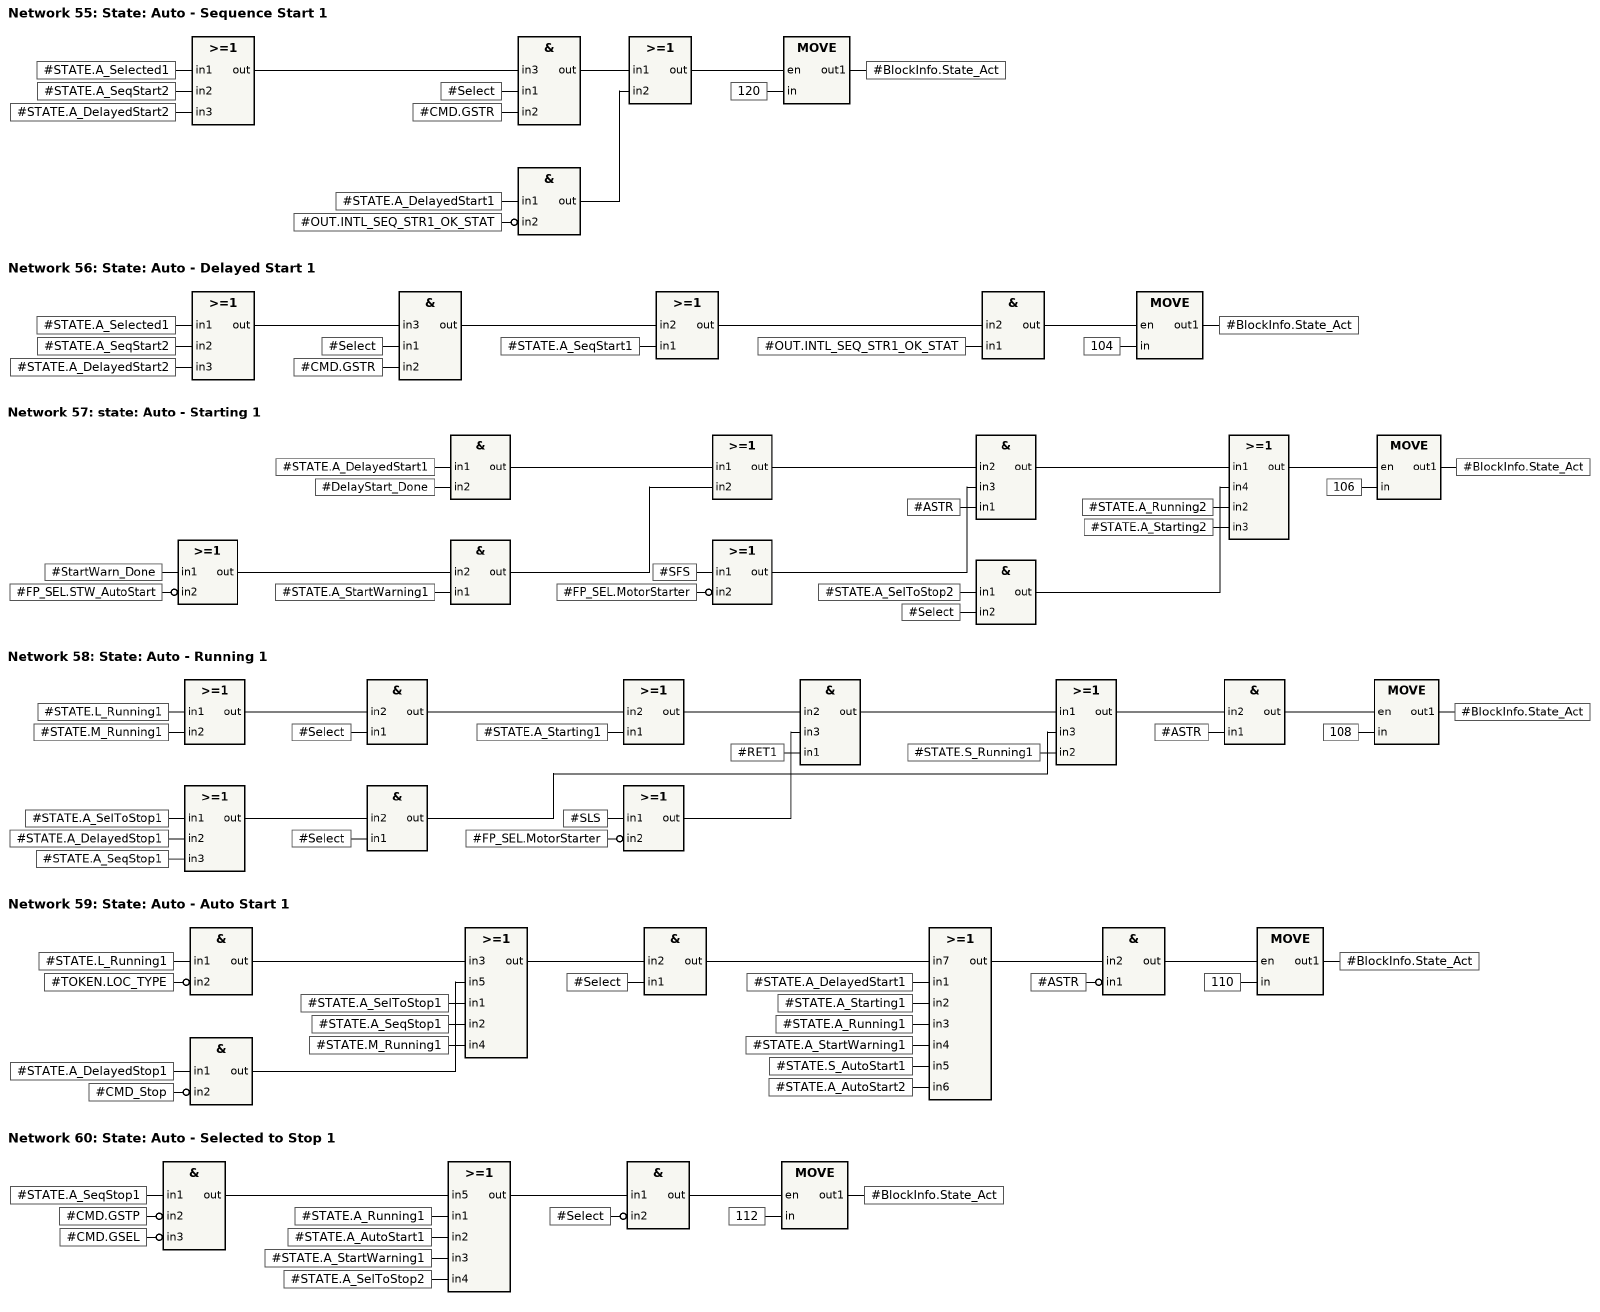
   IF ((#STATE.A_Selected1 OR #STATE.A_SeqStart2 OR #STATE.A_DelayedStart2) AND #Select AND #CMD.GSTR) OR (#STATE.A_DelayedStart1 AND NOT #OUT.INTL_SEQ_STR1_OK_STAT) THEN
       #BlockInfo.State_Act := 120;
   END_IF;
END_REGION

REGION Network 56: State: Auto - Delayed Start 1
   IF (((#STATE.A_Selected1 OR #STATE.A_SeqStart2 OR #STATE.A_DelayedStart2) AND #Select AND #CMD.GSTR) OR #STATE.A_SeqStart1) AND #OUT.INTL_SEQ_STR1_OK_STAT THEN
       #BlockInfo.State_Act := 104;
   END_IF;
END_REGION

REGION Network 57: state: Auto - Starting 1
   // Build 029 - 23.Sep.2021 (SURAM-IN) SFS Logic Added- While Starting SFS should be healthy.
   IF (((#STATE.A_DelayedStart1 AND #DelayStart_Done) OR ((#StartWarn_Done OR NOT #FP_SEL.STW_AutoStart) AND #STATE.A_StartWarning1)) AND (#SFS OR NOT #FP_SEL.MotorStarter) AND #ASTR) OR (#STATE.A_SelToStop2 AND #Select) OR #STATE.A_Running2 OR #STATE.A_Starting2 THEN
       #BlockInfo.State_Act := 106;
   END_IF;
END_REGION

REGION Network 58: State: Auto - Running 1
   IF (((((#STATE.L_Running1 OR #STATE.M_Running1) AND #Select) OR #STATE.A_Starting1) AND (#SLS OR NOT #FP_SEL.MotorStarter) AND #RET1) OR ((#STATE.A_SelToStop1 OR #STATE.A_DelayedStop1 OR #STATE.A_SeqStop1) AND #Select) OR #STATE.S_Running1) AND #ASTR THEN
       #BlockInfo.State_Act := 108;
   END_IF;
END_REGION

REGION Network 59: State: Auto - Auto Start 1
   // Build 003 - 1.July.2019 (EXTBOB): Add LOC_TYPE to L_Running1 condition
   // Build 006 - 29 Aug 2019 (EXTBOB) : Select & GSTR logic removed to make state machine to go to Seq_Start state when ASTR=0 & SEQ_START_INTL=0 during GSTR
   IF ((((#STATE.L_Running1 AND NOT #TOKEN.LOC_TYPE) OR (#STATE.A_DelayedStop1 AND NOT #CMD_Stop) OR #STATE.A_SelToStop1 OR #STATE.A_SeqStop1 OR #STATE.M_Running1) AND #Select) OR #STATE.A_DelayedStart1 OR #STATE.A_Starting1 OR #STATE.A_Running1 OR #STATE.A_StartWarning1 OR #STATE.S_AutoStart1 OR #STATE.A_AutoStart2) AND NOT #ASTR THEN
       #BlockInfo.State_Act := 110;
   END_IF;
END_REGION

REGION Network 60: State: Auto - Selected to Stop 1
   // Build 002 - 25 March 2019 : A_SeqStop1 with GSTP condition added
   // Build 004 - 11 Jul 2019 (EXTBOB) : GSEL added to A_SeqStop1 with GSTP condition to move to Selected to Stop state from Seq stop state if group stop timer ompletes
   IF ((#STATE.A_SeqStop1 AND NOT #CMD.GSTP AND NOT #CMD.GSEL) OR #STATE.A_Running1 OR #STATE.A_AutoStart1 OR #STATE.A_StartWarning1 OR #STATE.A_SelToStop2) AND NOT #Select THEN
       #BlockInfo.State_Act := 112;
   END_IF;
END_REGION

REGION Network 61: State: Auto - Sequence Stop 1
   // Build 002 - 25 March 2019 : A_SeqStop2 flag added
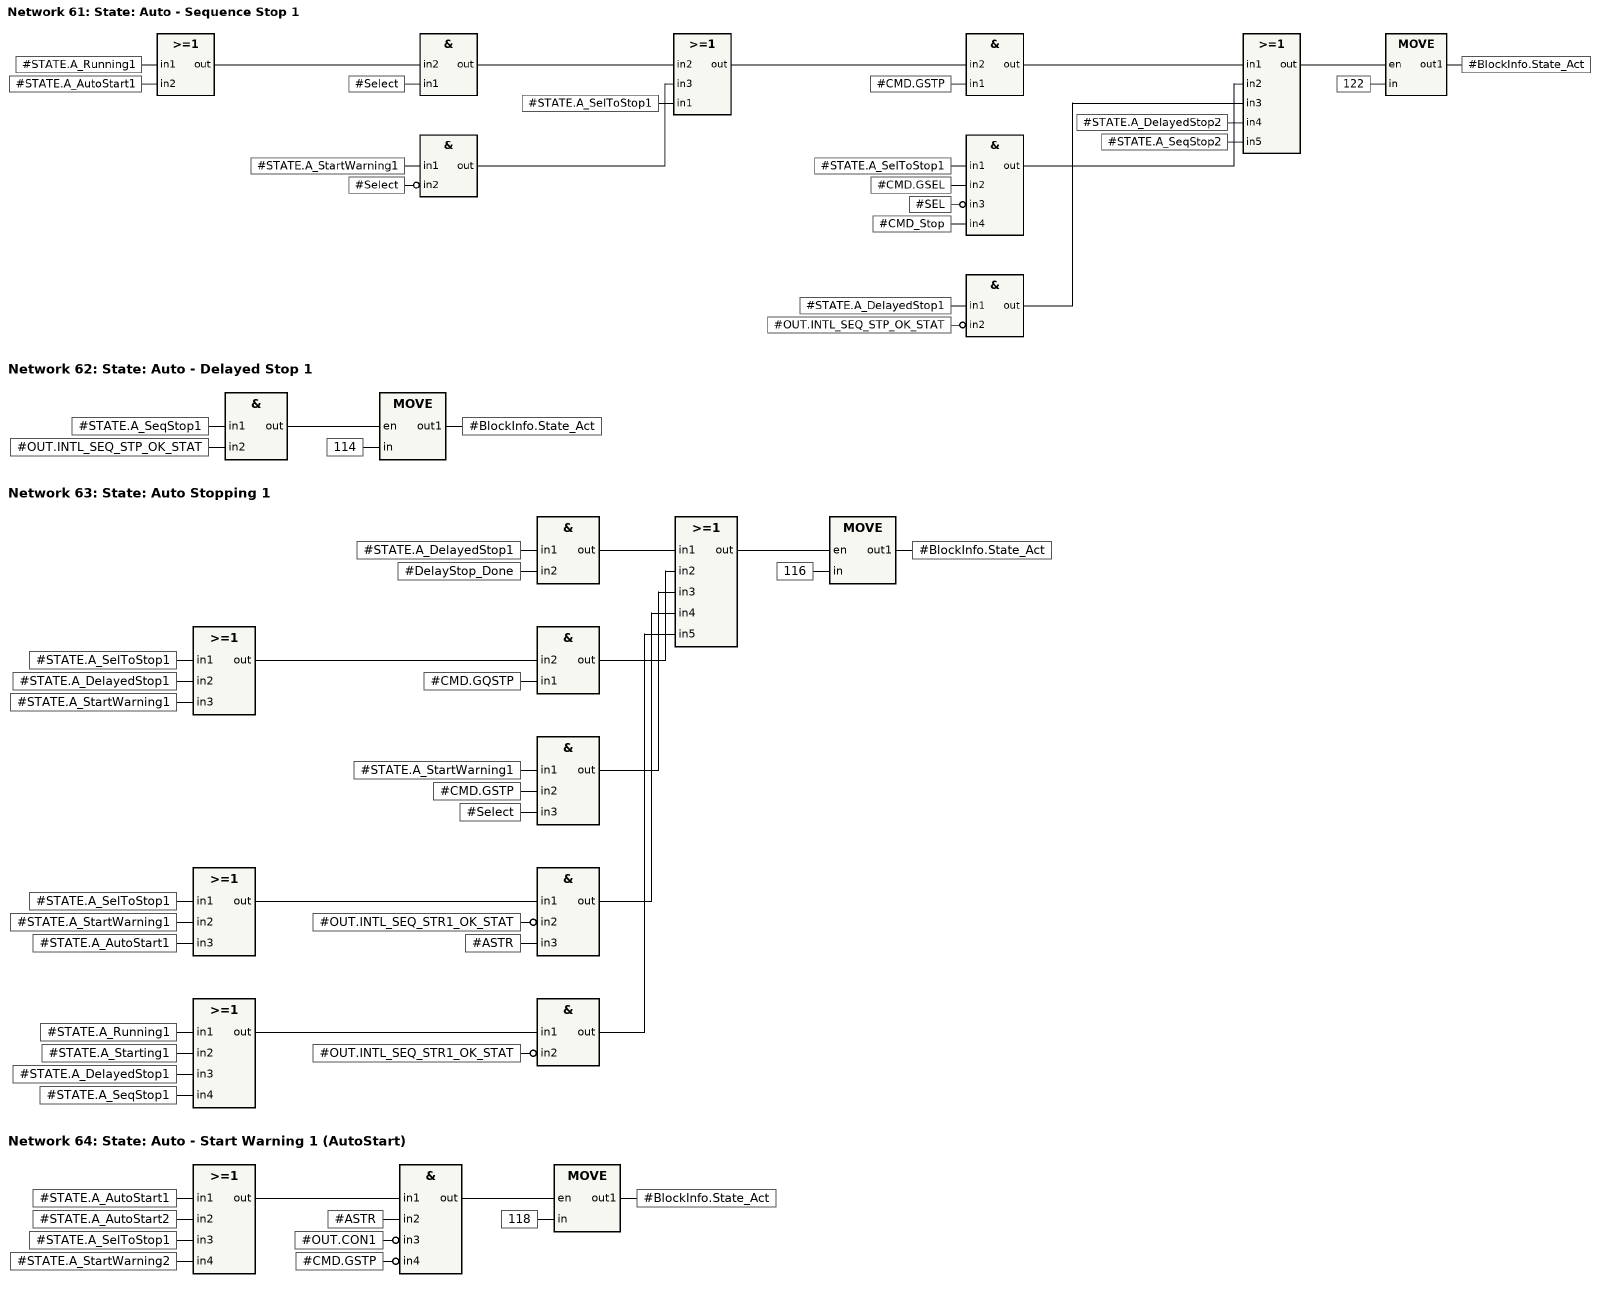
   IF ((((#STATE.A_Running1 OR #STATE.A_AutoStart1) AND #Select) OR (#STATE.A_StartWarning1 AND NOT #Select) OR #STATE.A_SelToStop1) AND #CMD.GSTP) OR (#STATE.A_SelToStop1 AND #CMD.GSEL AND NOT #SEL AND #CMD_Stop) OR (#STATE.A_DelayedStop1 AND NOT #OUT.INTL_SEQ_STP_OK_STAT) OR #STATE.A_DelayedStop2 OR #STATE.A_SeqStop2 THEN
       #BlockInfo.State_Act := 122;
   END_IF;
END_REGION

REGION Network 62: State: Auto - Delayed Stop 1
   IF #STATE.A_SeqStop1 AND #OUT.INTL_SEQ_STP_OK_STAT THEN #BlockInfo.State_Act := 114; END_IF;
END_REGION

REGION Network 63: State: Auto Stopping 1
   IF (#STATE.A_DelayedStop1 AND #DelayStop_Done) OR ((#STATE.A_SelToStop1 OR #STATE.A_DelayedStop1 OR #STATE.A_StartWarning1) AND #CMD.GQSTP) OR (#STATE.A_StartWarning1 AND #CMD.GSTP AND #Select) OR ((#STATE.A_SelToStop1 OR #STATE.A_StartWarning1 OR #STATE.A_AutoStart1) AND NOT #OUT.INTL_SEQ_STR1_OK_STAT AND #ASTR) OR ((#STATE.A_Running1 OR #STATE.A_Starting1 OR #STATE.A_DelayedStop1 OR #STATE.A_SeqStop1) AND NOT #OUT.INTL_SEQ_STR1_OK_STAT) THEN
       #BlockInfo.State_Act := 116;
   END_IF;
END_REGION

REGION Network 64: State: Auto - Start Warning 1 (AutoStart)
   IF (#STATE.A_AutoStart1 OR #STATE.A_AutoStart2 OR #STATE.A_SelToStop1 OR #STATE.A_StartWarning2) AND #ASTR AND NOT #OUT.CON1 AND NOT #CMD.GSTP THEN
       #BlockInfo.State_Act := 118;
   END_IF;
END_REGION

REGION Network 65
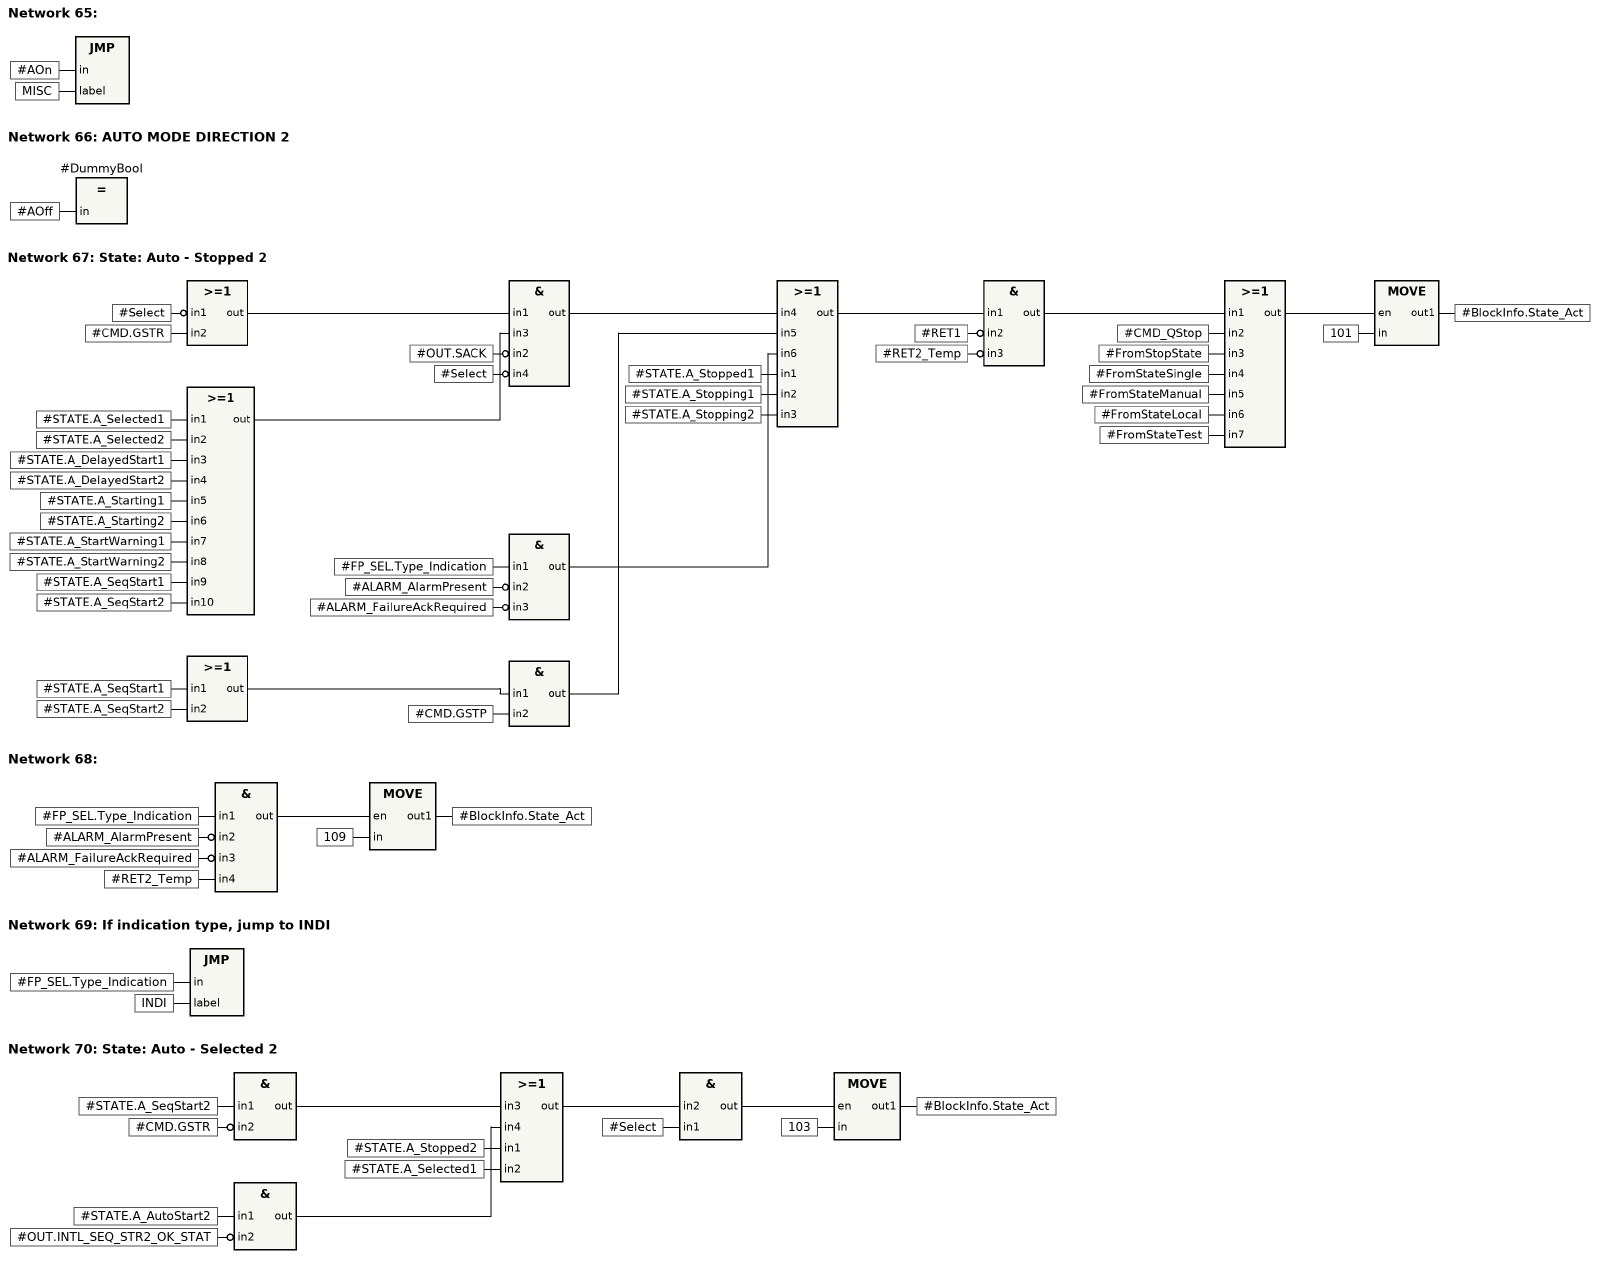
   IF #AOn THEN GOTO MISC; END_IF;
END_REGION

REGION Network 66: AUTO MODE DIRECTION 2
   AUT2:
   #DummyBool := #AOff;
END_REGION

REGION Network 67: State: Auto - Stopped 2
   IF ((((NOT #Select OR #CMD.GSTR) AND (#STATE.A_Selected1 OR #STATE.A_Selected2 OR #STATE.A_DelayedStart1 OR #STATE.A_DelayedStart2 OR #STATE.A_Starting1 OR #STATE.A_Starting2 OR #STATE.A_StartWarning1 OR #STATE.A_StartWarning2 OR #STATE.A_SeqStart1 OR #STATE.A_SeqStart2) AND NOT #OUT.SACK AND NOT #Select) OR ((#STATE.A_SeqStart1 OR #STATE.A_SeqStart2) AND #CMD.GSTP) OR (#FP_SEL.Type_Indication AND NOT #ALARM_AlarmPresent AND NOT #ALARM_FailureAckRequired) OR #STATE.A_Stopped1 OR #STATE.A_Stopping1 OR #STATE.A_Stopping2) AND NOT #RET1 AND NOT #RET2_Temp) OR #CMD_QStop OR #FromStopState OR #FromStateSingle OR #FromStateManual OR #FromStateLocal OR #FromStateTest THEN
       #BlockInfo.State_Act := 101;
   END_IF;
END_REGION

REGION Network 68
   IF #FP_SEL.Type_Indication AND NOT #ALARM_AlarmPresent AND NOT #ALARM_FailureAckRequired AND #RET2_Temp THEN
       #BlockInfo.State_Act := 109;
   END_IF;
END_REGION

REGION Network 69: If indication type, jump to INDI
   IF #FP_SEL.Type_Indication THEN GOTO INDI; END_IF;
END_REGION

REGION Network 70: State: Auto - Selected 2
   // Build 002 - 25 March 2019 : AutoSatrt2 with SeqStart Interlock condition added
   IF ((#STATE.A_SeqStart2 AND NOT #CMD.GSTR) OR (#STATE.A_AutoStart2 AND NOT #OUT.INTL_SEQ_STR2_OK_STAT) OR #STATE.A_Stopped2 OR #STATE.A_Selected1) AND #Select THEN
       #BlockInfo.State_Act := 103;
   END_IF;
END_REGION

REGION Network 71: State: Auto - Sequence Start 2
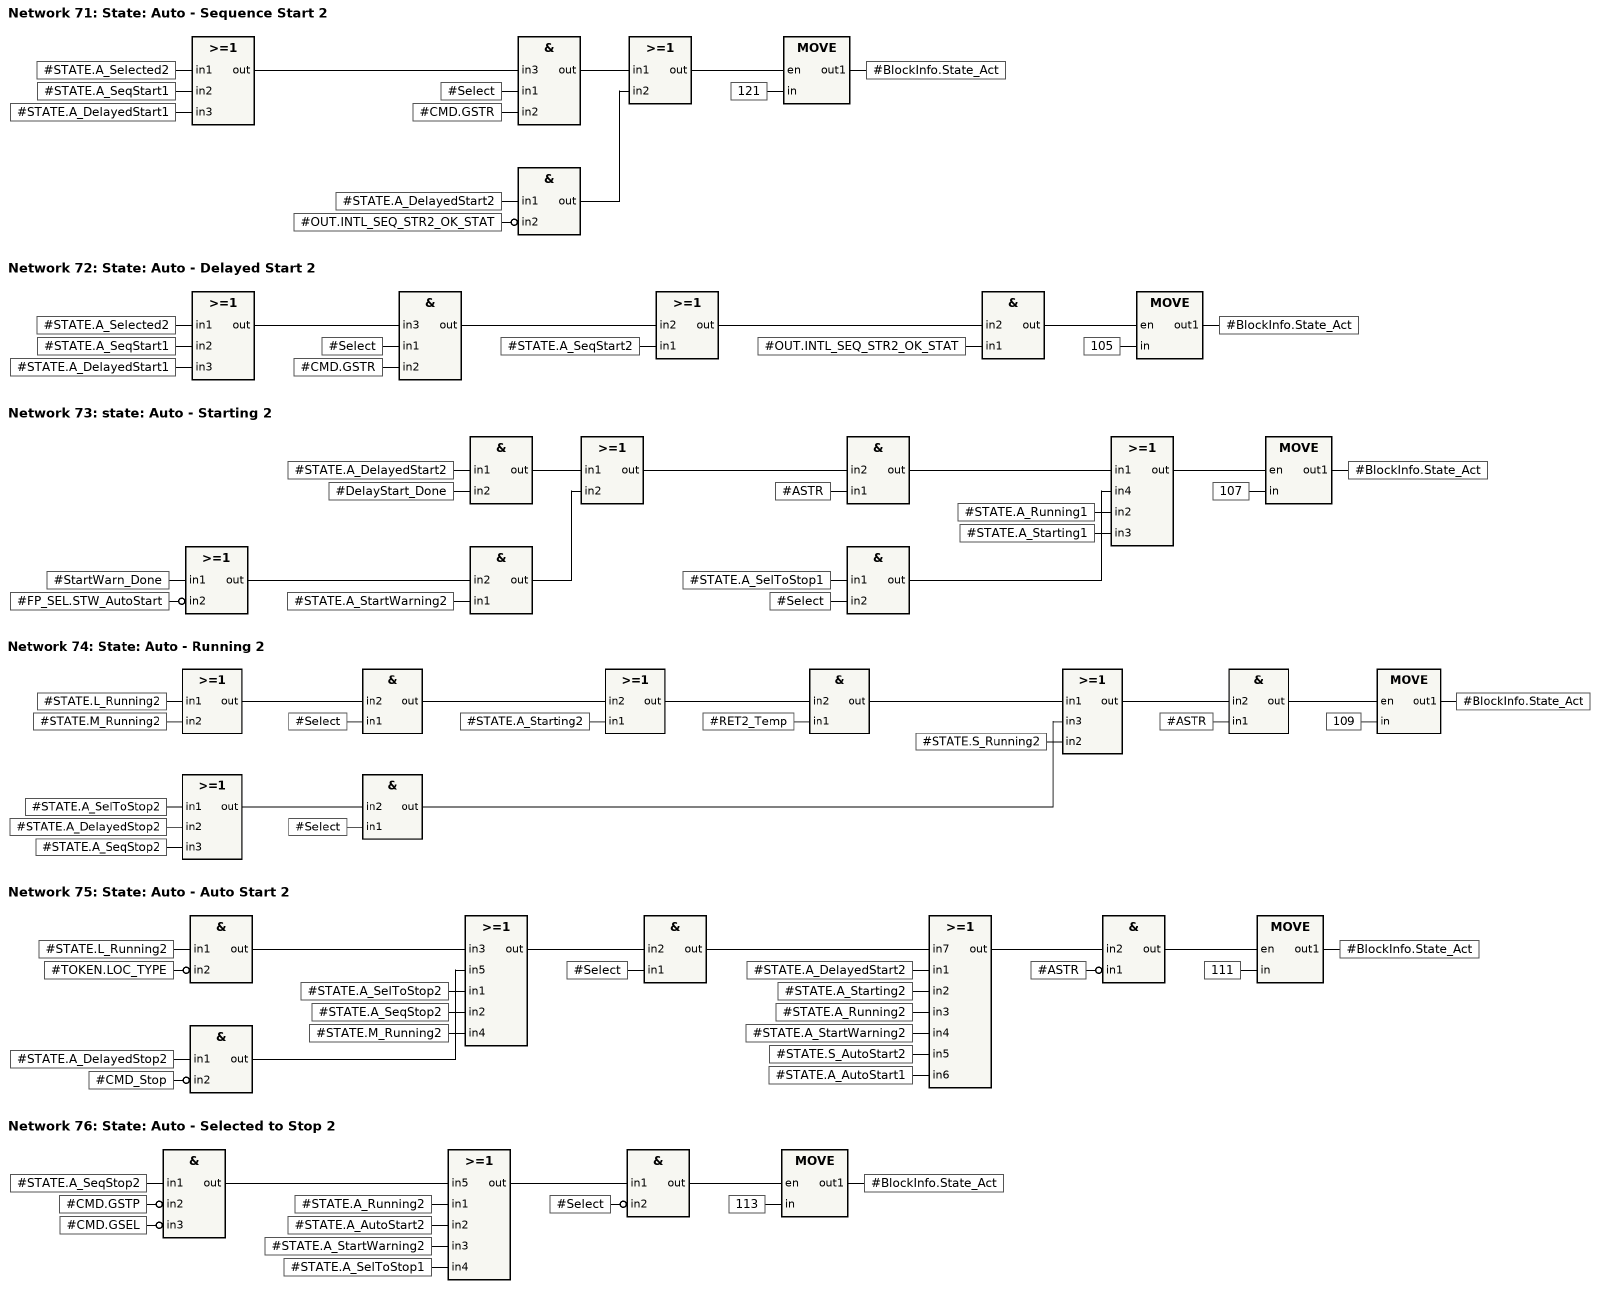
   IF ((#STATE.A_Selected2 OR #STATE.A_SeqStart1 OR #STATE.A_DelayedStart1) AND #Select AND #CMD.GSTR) OR (#STATE.A_DelayedStart2 AND NOT #OUT.INTL_SEQ_STR2_OK_STAT) THEN
       #BlockInfo.State_Act := 121;
   END_IF;
END_REGION

REGION Network 72: State: Auto - Delayed Start 2
   IF (((#STATE.A_Selected2 OR #STATE.A_SeqStart1 OR #STATE.A_DelayedStart1) AND #Select AND #CMD.GSTR) OR #STATE.A_SeqStart2) AND #OUT.INTL_SEQ_STR2_OK_STAT THEN
       #BlockInfo.State_Act := 105;
   END_IF;
END_REGION

REGION Network 73: state: Auto - Starting 2
   IF (((#STATE.A_DelayedStart2 AND #DelayStart_Done) OR ((#StartWarn_Done OR NOT #FP_SEL.STW_AutoStart) AND #STATE.A_StartWarning2)) AND #ASTR) OR (#STATE.A_SelToStop1 AND #Select) OR #STATE.A_Running1 OR #STATE.A_Starting1 THEN
       #BlockInfo.State_Act := 107;
   END_IF;
END_REGION

REGION Network 74: State: Auto - Running 2
   IF (((((#STATE.L_Running2 OR #STATE.M_Running2) AND #Select) OR #STATE.A_Starting2) AND #RET2_Temp) OR ((#STATE.A_SelToStop2 OR #STATE.A_DelayedStop2 OR #STATE.A_SeqStop2) AND #Select) OR #STATE.S_Running2) AND #ASTR THEN
       #BlockInfo.State_Act := 109;
   END_IF;
END_REGION

REGION Network 75: State: Auto - Auto Start 2
   // Build 003 - 1.July.2019 (EXTBOB): Add LOC_TYPE to L_Running2 condition
   // Build 006 - 29 Aug 2019 (EXTBOB) : Select & GSTR logic removed to make state machine to go to Seq_Start state when ASTR=0 & SEQ_START_INTL=0 during GSTR
   IF ((((#STATE.L_Running2 AND NOT #TOKEN.LOC_TYPE) OR (#STATE.A_DelayedStop2 AND NOT #CMD_Stop) OR #STATE.A_SelToStop2 OR #STATE.A_SeqStop2 OR #STATE.M_Running2) AND #Select) OR #STATE.A_DelayedStart2 OR #STATE.A_Starting2 OR #STATE.A_Running2 OR #STATE.A_StartWarning2 OR #STATE.S_AutoStart2 OR #STATE.A_AutoStart1) AND NOT #ASTR THEN
       #BlockInfo.State_Act := 111;
   END_IF;
END_REGION

REGION Network 76: State: Auto - Selected to Stop 2
   // Build 002 - 25 March 2019 : A_SeqStop2 with GSTP condition added
   // Build 004 - 11 Jul 2019 (EXTBOB) : GSEL added to A_SeqStop2 with GSTP condition to move to Selected to Stop state from Seq stop state if group stop timer ompletes
   IF ((#STATE.A_SeqStop2 AND NOT #CMD.GSTP AND NOT #CMD.GSEL) OR #STATE.A_Running2 OR #STATE.A_AutoStart2 OR #STATE.A_StartWarning2 OR #STATE.A_SelToStop1) AND NOT #Select THEN
       #BlockInfo.State_Act := 113;
   END_IF;
END_REGION

REGION Network 77: State: Auto - Sequence Stop 2
   // Build 002 - 25 March 2019 : A_SeqStop1 flag added
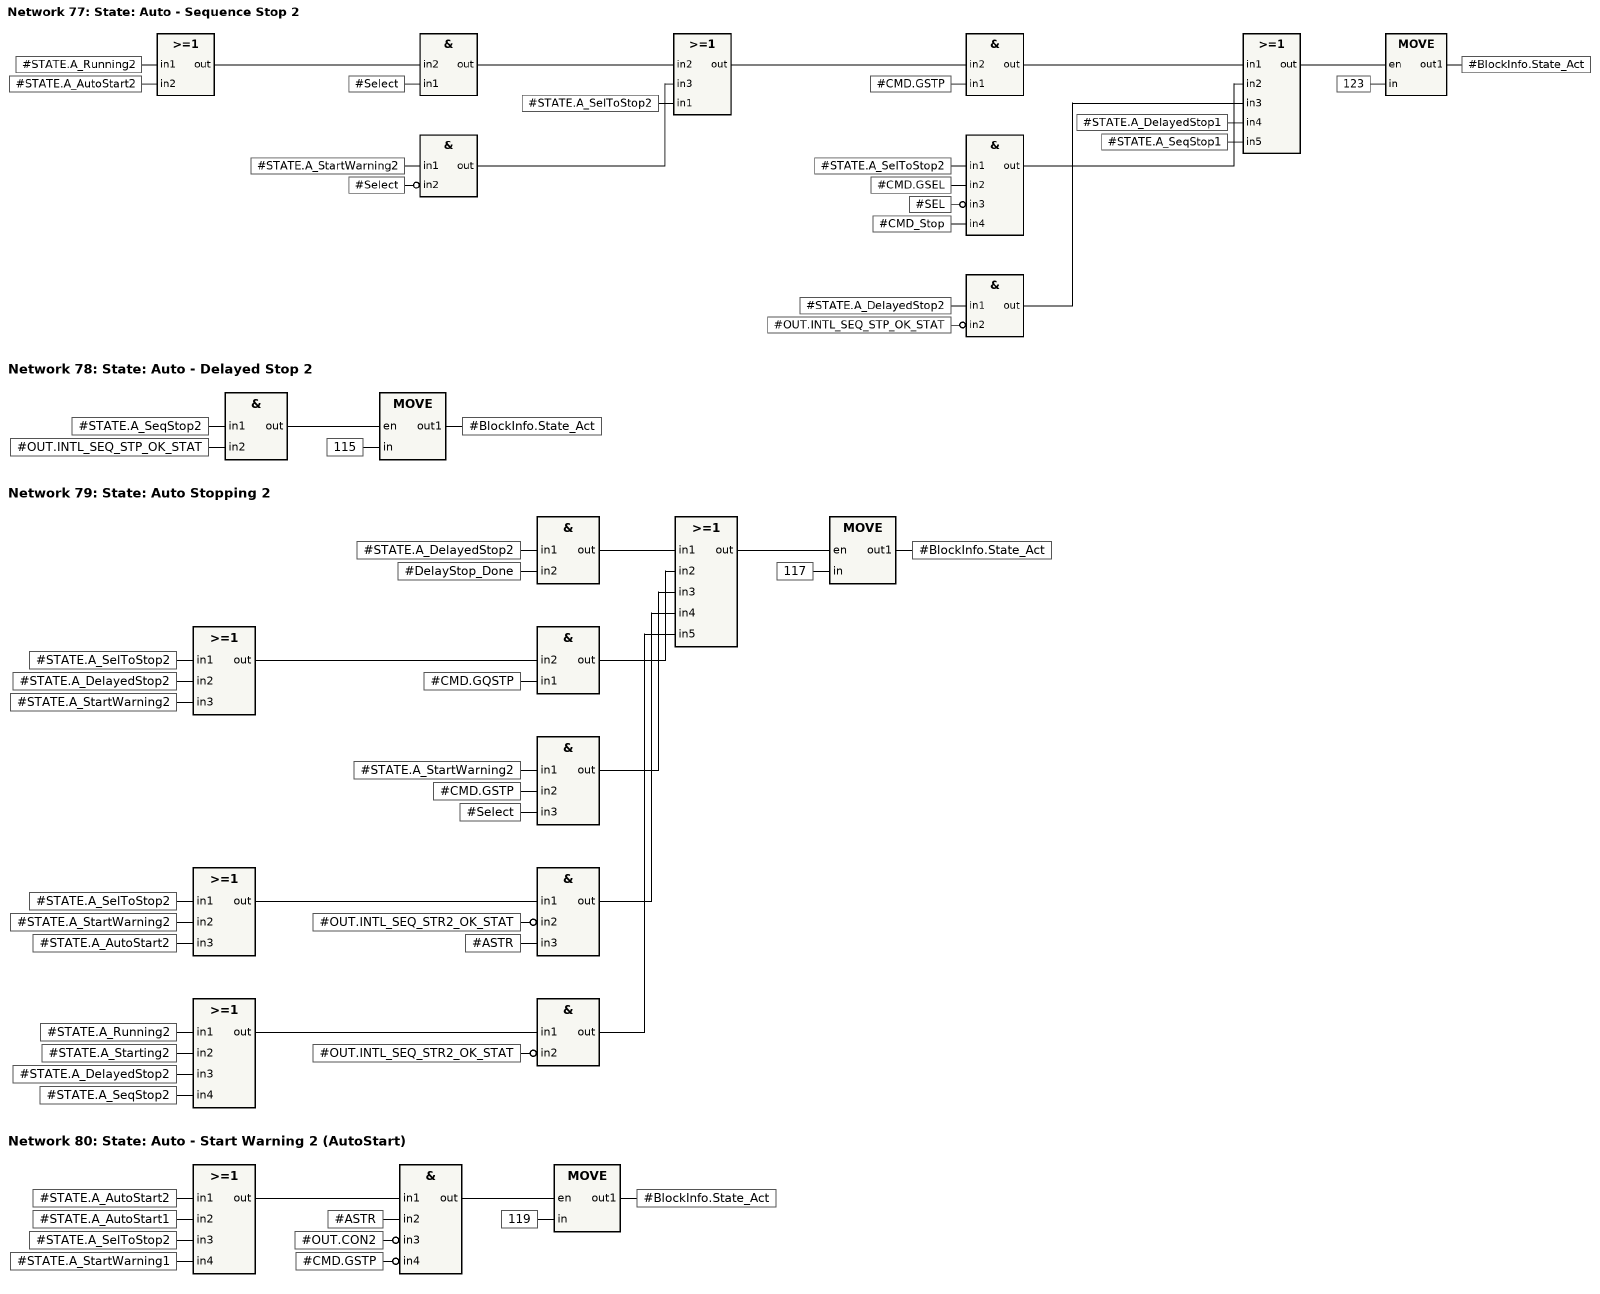
   IF ((((#STATE.A_Running2 OR #STATE.A_AutoStart2) AND #Select) OR (#STATE.A_StartWarning2 AND NOT #Select) OR #STATE.A_SelToStop2) AND #CMD.GSTP) OR (#STATE.A_SelToStop2 AND #CMD.GSEL AND NOT #SEL AND #CMD_Stop) OR (#STATE.A_DelayedStop2 AND NOT #OUT.INTL_SEQ_STP_OK_STAT) OR #STATE.A_DelayedStop1 OR #STATE.A_SeqStop1 THEN
       #BlockInfo.State_Act := 123;
   END_IF;
END_REGION

REGION Network 78: State: Auto - Delayed Stop 2
   IF #STATE.A_SeqStop2 AND #OUT.INTL_SEQ_STP_OK_STAT THEN #BlockInfo.State_Act := 115; END_IF;
END_REGION

REGION Network 79: State: Auto Stopping 2
   IF (#STATE.A_DelayedStop2 AND #DelayStop_Done) OR ((#STATE.A_SelToStop2 OR #STATE.A_DelayedStop2 OR #STATE.A_StartWarning2) AND #CMD.GQSTP) OR (#STATE.A_StartWarning2 AND #CMD.GSTP AND #Select) OR ((#STATE.A_SelToStop2 OR #STATE.A_StartWarning2 OR #STATE.A_AutoStart2) AND NOT #OUT.INTL_SEQ_STR2_OK_STAT AND #ASTR) OR ((#STATE.A_Running2 OR #STATE.A_Starting2 OR #STATE.A_DelayedStop2 OR #STATE.A_SeqStop2) AND NOT #OUT.INTL_SEQ_STR2_OK_STAT) THEN
       #BlockInfo.State_Act := 117;
   END_IF;
END_REGION

REGION Network 80: State: Auto - Start Warning 2 (AutoStart)
   IF (#STATE.A_AutoStart2 OR #STATE.A_AutoStart1 OR #STATE.A_SelToStop2 OR #STATE.A_StartWarning1) AND #ASTR AND NOT #OUT.CON2 AND NOT #CMD.GSTP THEN
       #BlockInfo.State_Act := 119;
   END_IF;
END_REGION

REGION Network 81
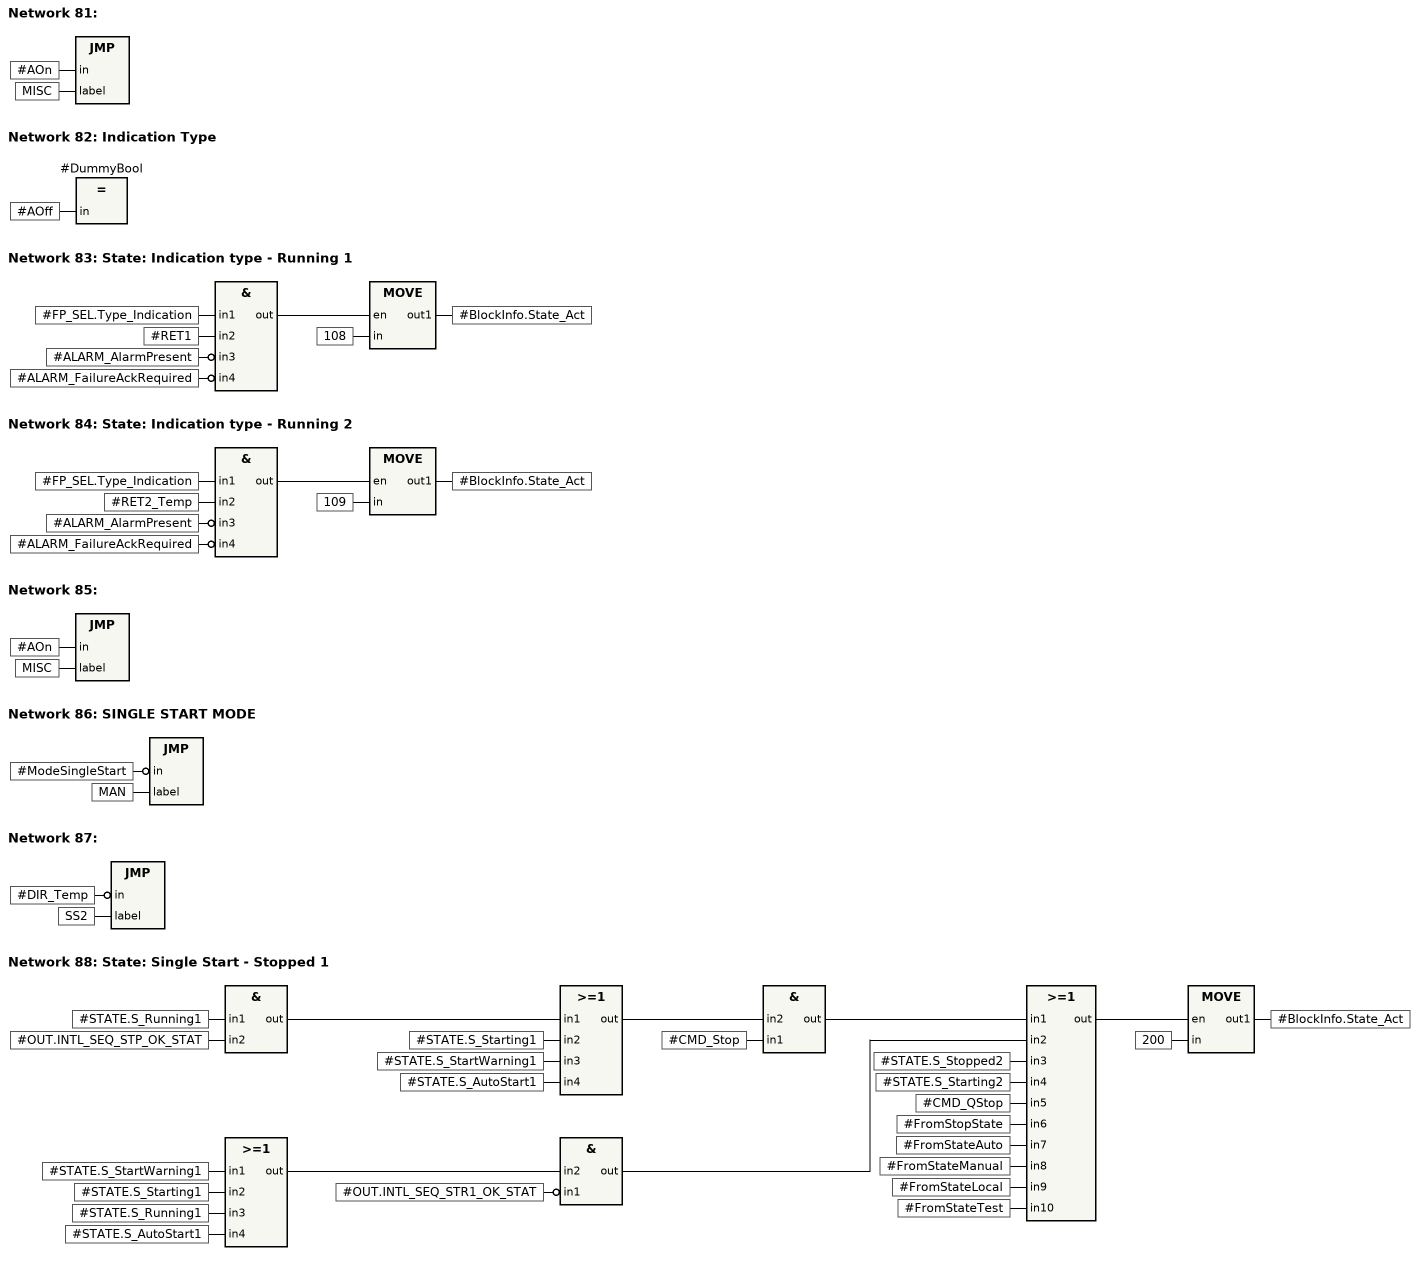
   IF #AOn THEN GOTO MISC; END_IF;
END_REGION

REGION Network 82: Indication Type
   INDI:
   #DummyBool := #AOff;
END_REGION

REGION Network 83: State: Indication type - Running 1
   IF #FP_SEL.Type_Indication AND #RET1 AND NOT #ALARM_AlarmPresent AND NOT #ALARM_FailureAckRequired THEN
       #BlockInfo.State_Act := 108;
   END_IF;
END_REGION

REGION Network 84: State: Indication type - Running 2
   IF #FP_SEL.Type_Indication AND #RET2_Temp AND NOT #ALARM_AlarmPresent AND NOT #ALARM_FailureAckRequired THEN
       #BlockInfo.State_Act := 109;
   END_IF;
END_REGION

REGION Network 85
   IF #AOn THEN GOTO MISC; END_IF;
END_REGION

REGION Network 86: SINGLE START MODE
   SS1:
   IF NOT #ModeSingleStart THEN GOTO MAN; END_IF;
END_REGION

REGION Network 87
   IF NOT #DIR_Temp THEN GOTO SS2; END_IF;
END_REGION

REGION Network 88: State: Single Start - Stopped 1
   // Build 002 - 25 March 2019 : AutoStart1 flag in Seq Start1 condition added
   IF (((#STATE.S_Running1 AND #OUT.INTL_SEQ_STP_OK_STAT) OR #STATE.S_Starting1 OR #STATE.S_StartWarning1 OR #STATE.S_AutoStart1) AND #CMD_Stop) OR ((#STATE.S_StartWarning1 OR #STATE.S_Starting1 OR #STATE.S_Running1 OR #STATE.S_AutoStart1) AND NOT #OUT.INTL_SEQ_STR1_OK_STAT) OR #STATE.S_Stopped2 OR #STATE.S_Starting2 OR #CMD_QStop OR #FromStopState OR #FromStateAuto OR #FromStateManual OR #FromStateLocal OR #FromStateTest THEN
       #BlockInfo.State_Act := 200;
   END_IF;
END_REGION

REGION Network 89: State: Single Start - Start Warning 1
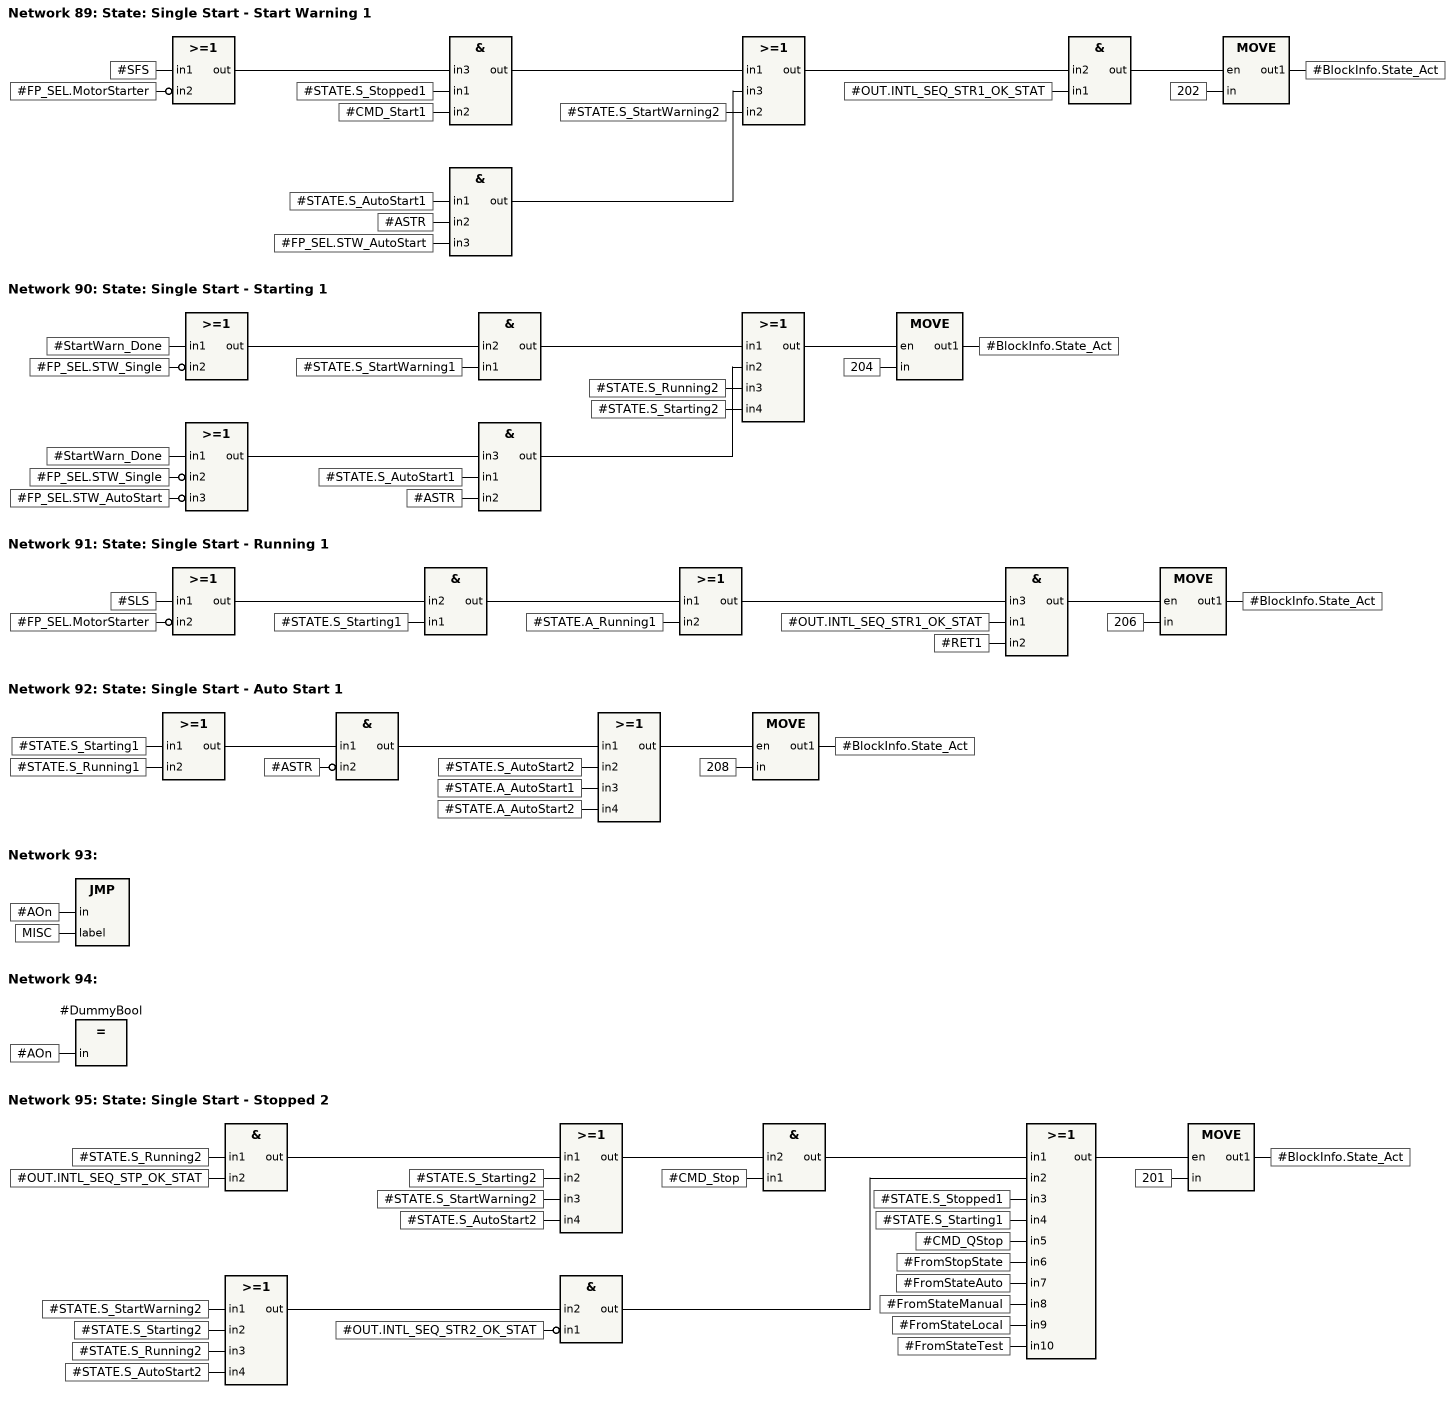
   IF (((#SFS OR NOT #FP_SEL.MotorStarter) AND #STATE.S_Stopped1 AND #CMD_Start1) OR (#STATE.S_AutoStart1 AND #ASTR AND #FP_SEL.STW_AutoStart) OR #STATE.S_StartWarning2) AND #OUT.INTL_SEQ_STR1_OK_STAT THEN
       #BlockInfo.State_Act := 202;
   END_IF;
END_REGION

REGION Network 90: State: Single Start - Starting 1
   IF ((#StartWarn_Done OR NOT #FP_SEL.STW_Single) AND #STATE.S_StartWarning1) OR ((#StartWarn_Done OR NOT #FP_SEL.STW_Single OR NOT #FP_SEL.STW_AutoStart) AND #STATE.S_AutoStart1 AND #ASTR) OR #STATE.S_Running2 OR #STATE.S_Starting2 THEN
       #BlockInfo.State_Act := 204;
   END_IF;
END_REGION

REGION Network 91: State: Single Start - Running 1
   IF (((#SLS OR NOT #FP_SEL.MotorStarter) AND #STATE.S_Starting1) OR #STATE.A_Running1) AND #OUT.INTL_SEQ_STR1_OK_STAT AND #RET1 THEN
       #BlockInfo.State_Act := 206;
   END_IF;
END_REGION

REGION Network 92: State: Single Start - Auto Start 1
   IF ((#STATE.S_Starting1 OR #STATE.S_Running1) AND NOT #ASTR) OR #STATE.S_AutoStart2 OR #STATE.A_AutoStart1 OR #STATE.A_AutoStart2 THEN
       #BlockInfo.State_Act := 208;
   END_IF;
END_REGION

REGION Network 93
   IF #AOn THEN GOTO MISC; END_IF;
END_REGION

REGION Network 94
   SS2:
   #DummyBool := #AOn;
END_REGION

REGION Network 95: State: Single Start - Stopped 2
   // Build 002 - 25 March 2019 : AutoStart2 flag in Seq Start2 condition added
   IF (((#STATE.S_Running2 AND #OUT.INTL_SEQ_STP_OK_STAT) OR #STATE.S_Starting2 OR #STATE.S_StartWarning2 OR #STATE.S_AutoStart2) AND #CMD_Stop) OR ((#STATE.S_StartWarning2 OR #STATE.S_Starting2 OR #STATE.S_Running2 OR #STATE.S_AutoStart2) AND NOT #OUT.INTL_SEQ_STR2_OK_STAT) OR #STATE.S_Stopped1 OR #STATE.S_Starting1 OR #CMD_QStop OR #FromStopState OR #FromStateAuto OR #FromStateManual OR #FromStateLocal OR #FromStateTest THEN
       #BlockInfo.State_Act := 201;
   END_IF;
END_REGION

REGION Network 96: State: Single Start - Start Warning 2
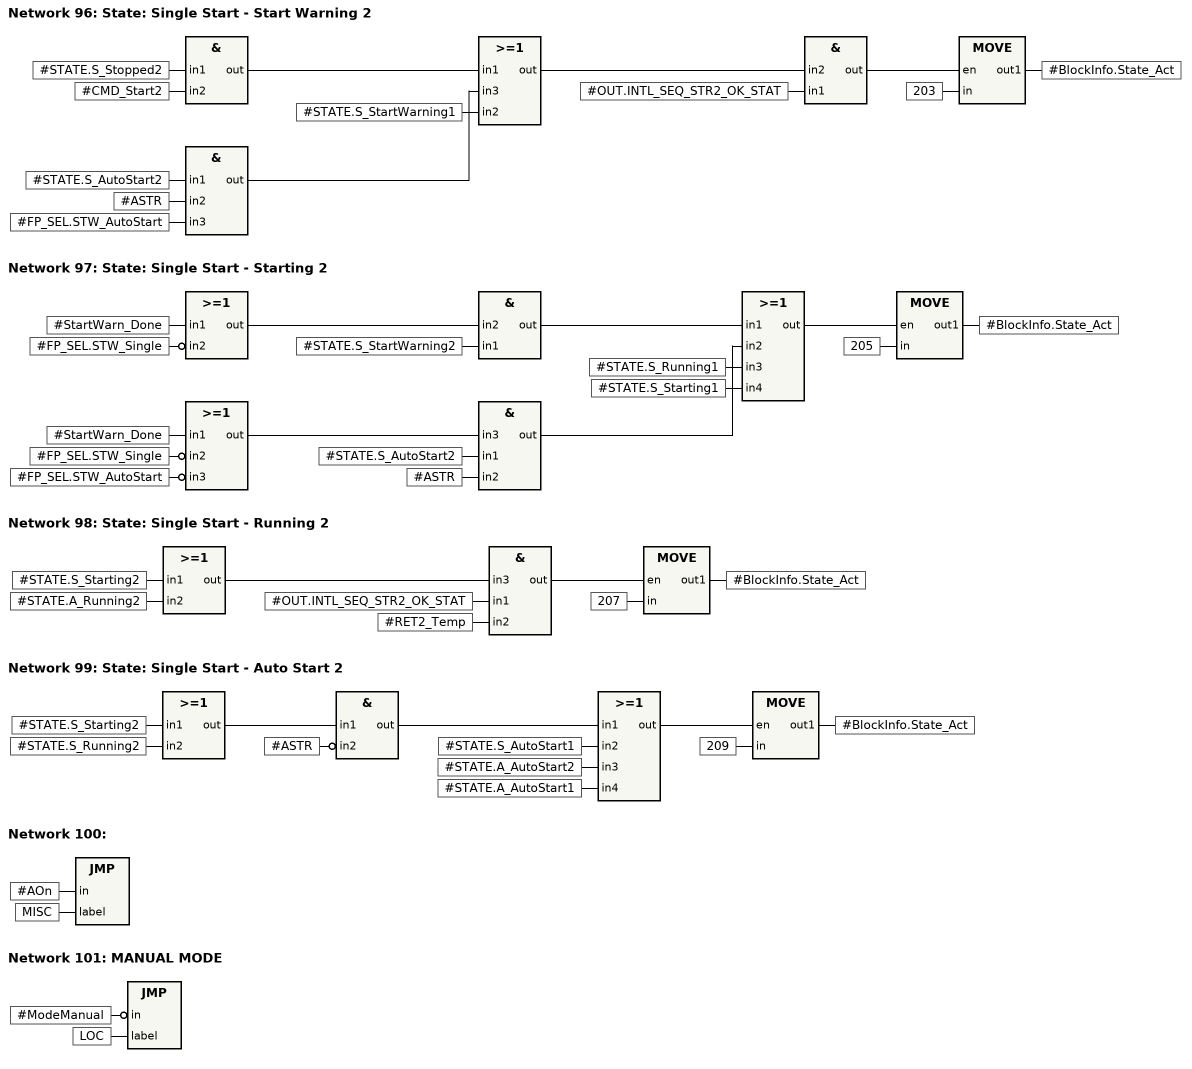
   IF ((#STATE.S_Stopped2 AND #CMD_Start2) OR (#STATE.S_AutoStart2 AND #ASTR AND #FP_SEL.STW_AutoStart) OR #STATE.S_StartWarning1) AND #OUT.INTL_SEQ_STR2_OK_STAT THEN
       #BlockInfo.State_Act := 203;
   END_IF;
END_REGION

REGION Network 97: State: Single Start - Starting 2
   IF ((#StartWarn_Done OR NOT #FP_SEL.STW_Single) AND #STATE.S_StartWarning2) OR ((#StartWarn_Done OR NOT #FP_SEL.STW_Single OR NOT #FP_SEL.STW_AutoStart) AND #STATE.S_AutoStart2 AND #ASTR) OR #STATE.S_Running1 OR #STATE.S_Starting1 THEN
       #BlockInfo.State_Act := 205;
   END_IF;
END_REGION

REGION Network 98: State: Single Start - Running 2
   IF (#STATE.S_Starting2 OR #STATE.A_Running2) AND #OUT.INTL_SEQ_STR2_OK_STAT AND #RET2_Temp THEN
       #BlockInfo.State_Act := 207;
   END_IF;
END_REGION

REGION Network 99: State: Single Start - Auto Start 2
   IF ((#STATE.S_Starting2 OR #STATE.S_Running2) AND NOT #ASTR) OR #STATE.S_AutoStart1 OR #STATE.A_AutoStart2 OR #STATE.A_AutoStart1 THEN
       #BlockInfo.State_Act := 209;
   END_IF;
END_REGION

REGION Network 100
   IF #AOn THEN GOTO MISC; END_IF;
END_REGION

REGION Network 101: MANUAL MODE
   MAN:
   IF NOT #ModeManual THEN GOTO LOC; END_IF;
END_REGION

REGION Network 102: State: Manual - Stopped
   // Build 013 - 21.Feb.2022 (SURAM-IN) FP_CMD.Start1,  FP_CMD.Start2 and FP_SEL.INCH_Man logic added for Inching in Manual Mode
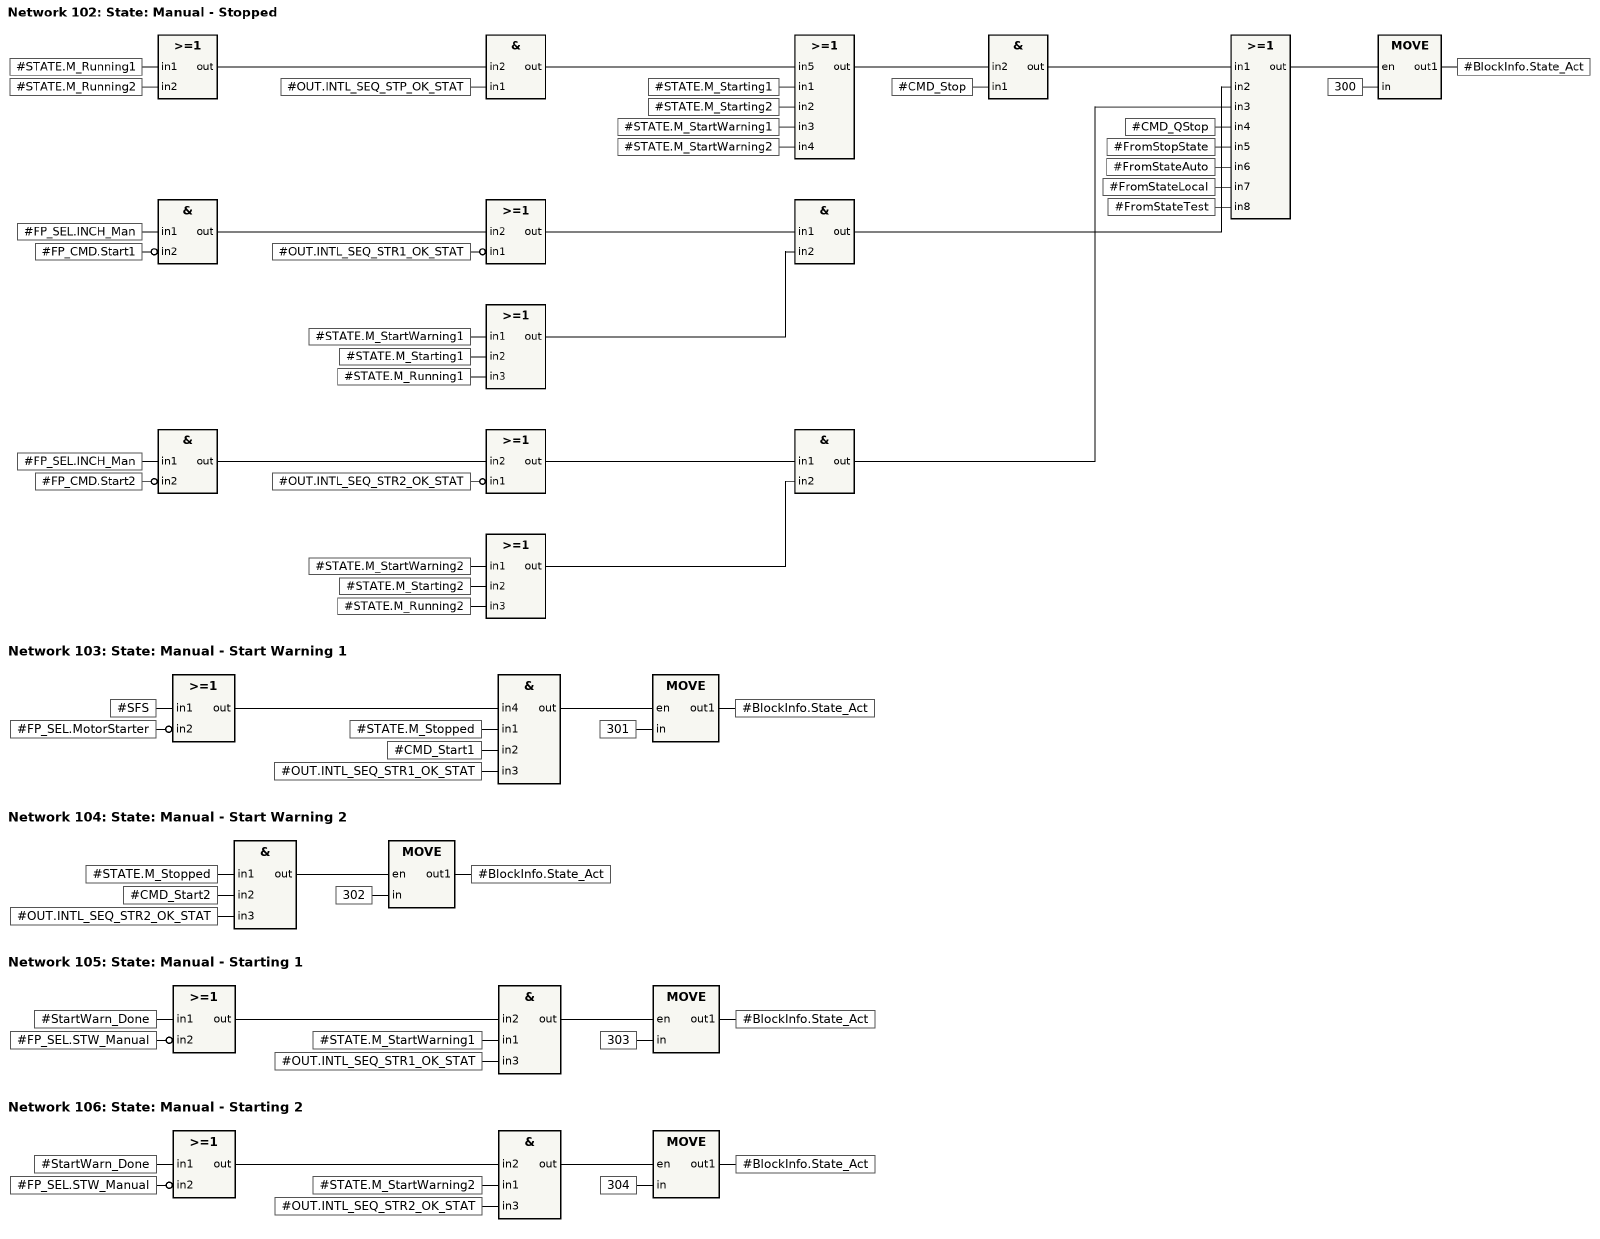
   IF ((((#STATE.M_Running1 OR #STATE.M_Running2) AND #OUT.INTL_SEQ_STP_OK_STAT) OR #STATE.M_Starting1 OR #STATE.M_Starting2 OR #STATE.M_StartWarning1 OR #STATE.M_StartWarning2) AND #CMD_Stop) OR (((#FP_SEL.INCH_Man AND NOT #FP_CMD.Start1) OR NOT #OUT.INTL_SEQ_STR1_OK_STAT) AND (#STATE.M_StartWarning1 OR #STATE.M_Starting1 OR #STATE.M_Running1)) OR (((#FP_SEL.INCH_Man AND NOT #FP_CMD.Start2) OR NOT #OUT.INTL_SEQ_STR2_OK_STAT) AND (#STATE.M_StartWarning2 OR #STATE.M_Starting2 OR #STATE.M_Running2)) OR #CMD_QStop OR #FromStopState OR #FromStateAuto OR #FromStateLocal OR #FromStateTest THEN
       #BlockInfo.State_Act := 300;
   END_IF;
END_REGION

REGION Network 103: State: Manual - Start Warning 1
   IF (#SFS OR NOT #FP_SEL.MotorStarter) AND #STATE.M_Stopped AND #CMD_Start1 AND #OUT.INTL_SEQ_STR1_OK_STAT THEN
       #BlockInfo.State_Act := 301;
   END_IF;
END_REGION

REGION Network 104: State: Manual - Start Warning 2
   IF #STATE.M_Stopped AND #CMD_Start2 AND #OUT.INTL_SEQ_STR2_OK_STAT THEN
       #BlockInfo.State_Act := 302;
   END_IF;
END_REGION

REGION Network 105: State: Manual - Starting 1
   IF (#StartWarn_Done OR NOT #FP_SEL.STW_Manual) AND #STATE.M_StartWarning1 AND #OUT.INTL_SEQ_STR1_OK_STAT THEN
       #BlockInfo.State_Act := 303;
   END_IF;
END_REGION

REGION Network 106: State: Manual - Starting 2
   IF (#StartWarn_Done OR NOT #FP_SEL.STW_Manual) AND #STATE.M_StartWarning2 AND #OUT.INTL_SEQ_STR2_OK_STAT THEN
       #BlockInfo.State_Act := 304;
   END_IF;
END_REGION

REGION Network 107: State: Manual - Running 1
